  PROC DrawPart12()
    MoveL Offs(pOrigin,259.21,32.84,0.00),v40,z0,tPen\WObj:=wPaper;
    MoveL Offs(pOrigin,259.99,30.50,0.00),v40,z0,tPen\WObj:=wPaper;
    MoveL Offs(pOrigin,259.77,29.44,0.00),v40,z0,tPen\WObj:=wPaper;
    MoveL Offs(pOrigin,259.77,29.44,0.00),v40,z0,tPen\WObj:=wPaper;
    MoveL Offs(pOrigin,257.23,29.30,0.00),v40,z0,tPen\WObj:=wPaper;
    MoveL Offs(pOrigin,255.74,30.50,0.00),v40,z0,tPen\WObj:=wPaper;
    MoveL Offs(pOrigin,255.31,31.35,0.00),v40,z0,tPen\WObj:=wPaper;
    MoveL Offs(pOrigin,255.38,31.99,0.00),v40,z0,tPen\WObj:=wPaper;
    MoveL Offs(pOrigin,256.16,32.84,0.00),v40,z0,tPen\WObj:=wPaper;
    MoveL Offs(pOrigin,257.65,33.83,0.00),v40,z0,tPen\WObj:=wPaper;
    MoveL Offs(pOrigin,258.50,33.90,0.00),v40,z0,tPen\WObj:=wPaper;
    MoveL Offs(pOrigin,257.86,34.01,0.00),v40,z0,tPen\WObj:=wPaper;
    MoveL Offs(pOrigin,256.16,34.01,0.00),v40,z0,tPen\WObj:=wPaper;
    MoveL Offs(pOrigin,256.16,32.95,0.00),v40,z0,tPen\WObj:=wPaper;
    MoveL Offs(pOrigin,254.46,32.95,0.00),v40,z0,tPen\WObj:=wPaper;
    MoveL Offs(pOrigin,254.51,32.62,0.00),v40,z0,tPen\WObj:=wPaper;
    MoveL Offs(pOrigin,254.51,29.86,0.00),v40,z0,tPen\WObj:=wPaper;
    MoveL Offs(pOrigin,254.26,29.05,0.00),v40,z0,tPen\WObj:=wPaper;
    MoveL Offs(pOrigin,255.91,30.70,0.00),v40,z0,tPen\WObj:=wPaper;
    MoveL Offs(pOrigin,255.52,30.84,0.00),v40,z0,tPen\WObj:=wPaper;
    MoveL Offs(pOrigin,245.54,30.84,0.00),v40,z0,tPen\WObj:=wPaper;
    MoveL Offs(pOrigin,245.27,30.52,0.00),v40,z0,tPen\WObj:=wPaper;
    MoveL Offs(pOrigin,246.78,32.02,0.00),v40,z0,tPen\WObj:=wPaper;
    MoveL Offs(pOrigin,246.18,31.90,0.00),v40,z0,tPen\WObj:=wPaper;
    MoveL Offs(pOrigin,244.69,31.90,0.00),v40,z0,tPen\WObj:=wPaper;
    MoveL Offs(pOrigin,244.53,31.26,0.00),v40,z0,tPen\WObj:=wPaper;
    MoveL Offs(pOrigin,246.03,32.77,0.00),v40,z0,tPen\WObj:=wPaper;
    MoveL Offs(pOrigin,245.54,32.95,0.00),v40,z0,tPen\WObj:=wPaper;
    MoveL Offs(pOrigin,244.26,32.95,0.00),v40,z0,tPen\WObj:=wPaper;
    MoveL Offs(pOrigin,243.64,33.36,0.00),v40,z0,tPen\WObj:=wPaper;
    MoveL Offs(pOrigin,259.41,49.14,0.00),v40,z0,tPen\WObj:=wPaper;
    MoveL Offs(pOrigin,259.73,49.65,0.00),v40,z0,tPen\WObj:=wPaper;
    MoveL Offs(pOrigin,261.69,47.70,0.00),v40,z0,tPen\WObj:=wPaper;
    MoveL Offs(pOrigin,261.06,47.79,0.00),v40,z0,tPen\WObj:=wPaper;
    MoveL Offs(pOrigin,266.77,53.50,0.00),v40,z0,tPen\WObj:=wPaper;
    MoveL Offs(pOrigin,266.16,53.68,0.00),v40,z0,tPen\WObj:=wPaper;
    MoveL Offs(pOrigin,268.42,51.42,0.00),v40,z0,tPen\WObj:=wPaper;
    MoveL Offs(pOrigin,268.26,52.01,0.00),v40,z0,tPen\WObj:=wPaper;
    MoveL Offs(pOrigin,274.12,57.87,0.00),v40,z0,tPen\WObj:=wPaper;
    MoveL Offs(pOrigin,273.16,58.30,0.00),v40,z0,tPen\WObj:=wPaper;
    MoveL Offs(pOrigin,272.10,58.30,0.00),v40,z0,tPen\WObj:=wPaper;
    MoveL Offs(pOrigin,272.31,58.76,0.00),v40,z0,tPen\WObj:=wPaper;
    MoveL Offs(pOrigin,272.10,59.19,0.00),v40,z0,tPen\WObj:=wPaper;
    MoveL Offs(pOrigin,272.31,58.76,0.00),v40,z0,tPen\WObj:=wPaper;
    MoveL Offs(pOrigin,272.52,59.35,0.00),v40,z0,tPen\WObj:=wPaper;
    MoveL Offs(pOrigin,271.46,59.35,0.00),v40,z0,tPen\WObj:=wPaper;
    MoveL Offs(pOrigin,271.89,60.41,0.00),v40,z0,tPen\WObj:=wPaper;
    MoveL Offs(pOrigin,270.82,60.41,0.00),v40,z0,tPen\WObj:=wPaper;
    MoveL Offs(pOrigin,271.04,61.10,0.00),v40,z0,tPen\WObj:=wPaper;
    MoveL Offs(pOrigin,272.95,57.49,0.00),v40,z0,tPen\WObj:=wPaper;
    MoveL Offs(pOrigin,272.95,57.49,0.00),v40,z0,tPen\WObj:=wPaper;
    MoveL Offs(pOrigin,272.67,55.58,0.00),v40,z0,tPen\WObj:=wPaper;
    MoveL Offs(pOrigin,271.04,55.43,0.00),v40,z0,tPen\WObj:=wPaper;
    MoveL Offs(pOrigin,268.06,60.46,0.00),v40,z0,tPen\WObj:=wPaper;
    MoveL Offs(pOrigin,268.06,60.46,0.00),v40,z0,tPen\WObj:=wPaper;
    MoveL Offs(pOrigin,268.91,61.53,0.00),v40,z0,tPen\WObj:=wPaper;
    MoveL Offs(pOrigin,270.97,61.31,0.00),v40,z0,tPen\WObj:=wPaper;
    MoveL Offs(pOrigin,271.25,62.59,0.00),v40,z0,tPen\WObj:=wPaper;
    MoveL Offs(pOrigin,276.77,65.28,0.00),v40,z0,tPen\WObj:=wPaper;
    MoveL Offs(pOrigin,281.45,67.05,0.00),v40,z0,tPen\WObj:=wPaper;
    MoveL Offs(pOrigin,283.58,67.26,0.00),v40,z0,tPen\WObj:=wPaper;
    MoveL Offs(pOrigin,286.12,66.48,0.00),v40,z0,tPen\WObj:=wPaper;
    MoveL Offs(pOrigin,292.71,62.94,0.00),v40,z0,tPen\WObj:=wPaper;
    MoveL Offs(pOrigin,300.36,60.46,0.00),v40,z0,tPen\WObj:=wPaper;
    MoveL Offs(pOrigin,304.61,59.61,0.00),v40,z0,tPen\WObj:=wPaper;
    MoveL Offs(pOrigin,312.26,60.25,0.00),v40,z0,tPen\WObj:=wPaper;
    MoveL Offs(pOrigin,315.45,59.47,0.00),v40,z0,tPen\WObj:=wPaper;
    MoveL Offs(pOrigin,317.58,57.49,0.00),v40,z0,tPen\WObj:=wPaper;
    MoveL Offs(pOrigin,320.27,53.45,0.00),v40,z0,tPen\WObj:=wPaper;
    MoveL Offs(pOrigin,320.41,52.60,0.00),v40,z0,tPen\WObj:=wPaper;
    MoveL Offs(pOrigin,321.68,51.54,0.00),v40,z0,tPen\WObj:=wPaper;
    MoveL Offs(pOrigin,322.25,49.20,0.00),v40,z0,tPen\WObj:=wPaper;
    MoveL Offs(pOrigin,322.25,49.20,0.00),v40,z0,tPen\WObj:=wPaper;
    MoveL Offs(pOrigin,322.67,48.35,0.00),v40,z0,tPen\WObj:=wPaper;
    MoveL Offs(pOrigin,322.25,47.92,0.00),v40,z0,tPen\WObj:=wPaper;
    MoveL Offs(pOrigin,322.25,47.92,0.00),v40,z0,tPen\WObj:=wPaper;
    MoveL Offs(pOrigin,322.89,44.53,0.00),v40,z0,tPen\WObj:=wPaper;
    MoveL Offs(pOrigin,322.89,42.40,0.00),v40,z0,tPen\WObj:=wPaper;
    MoveL Offs(pOrigin,322.89,42.40,0.00),v40,z0,tPen\WObj:=wPaper;
    MoveL Offs(pOrigin,323.52,41.76,0.00),v40,z0,tPen\WObj:=wPaper;
    MoveL Offs(pOrigin,323.45,40.70,0.00),v40,z0,tPen\WObj:=wPaper;
    MoveL Offs(pOrigin,322.89,40.28,0.00),v40,z0,tPen\WObj:=wPaper;
    MoveL Offs(pOrigin,322.89,40.28,0.00),v40,z0,tPen\WObj:=wPaper;
    MoveL Offs(pOrigin,322.46,40.70,0.00),v40,z0,tPen\WObj:=wPaper;
    MoveL Offs(pOrigin,322.46,41.97,0.00),v40,z0,tPen\WObj:=wPaper;
    MoveL Offs(pOrigin,322.89,42.40,0.00),v40,z0,tPen\WObj:=wPaper;
    MoveL Offs(pOrigin,322.76,42.29,0.00),v40,z0,tPen\WObj:=wPaper;
    MoveL Offs(pOrigin,324.86,44.39,0.00),v40,z0,tPen\WObj:=wPaper;
    MoveL Offs(pOrigin,325.36,45.25,0.00),v40,z0,tPen\WObj:=wPaper;
    MoveL Offs(pOrigin,319.80,50.81,0.00),v40,fine,tPen\WObj:=wPaper;
    MoveL Offs(pOrigin,319.80,50.81,6.00),v60,z5,tPen\WObj:=wPaper;
    MoveL Offs(pOrigin,321.14,51.12,6.00),vTravel,z5,tPen\WObj:=wPaper;
    MoveL Offs(pOrigin,321.14,51.12,0.00),v60,z0,tPen\WObj:=wPaper;
    MoveL Offs(pOrigin,322.94,52.93,0.00),v40,z0,tPen\WObj:=wPaper;
    MoveL Offs(pOrigin,322.46,53.02,0.00),v40,z0,tPen\WObj:=wPaper;
    MoveL Offs(pOrigin,320.98,53.02,0.00),v40,z0,tPen\WObj:=wPaper;
    MoveL Offs(pOrigin,320.34,52.39,0.00),v40,z0,tPen\WObj:=wPaper;
    MoveL Offs(pOrigin,320.90,50.26,0.00),v40,z0,tPen\WObj:=wPaper;
    MoveL Offs(pOrigin,321.61,49.20,0.00),v40,z0,tPen\WObj:=wPaper;
    MoveL Offs(pOrigin,321.61,49.20,0.00),v40,z0,tPen\WObj:=wPaper;
    MoveL Offs(pOrigin,321.61,48.14,0.00),v40,z0,tPen\WObj:=wPaper;
    MoveL Offs(pOrigin,322.25,47.92,0.00),v40,z0,tPen\WObj:=wPaper;
    MoveL Offs(pOrigin,321.87,47.38,0.00),v40,z0,tPen\WObj:=wPaper;
    MoveL Offs(pOrigin,323.83,49.33,0.00),v40,z0,tPen\WObj:=wPaper;
    MoveL Offs(pOrigin,324.75,48.85,0.00),v40,z0,tPen\WObj:=wPaper;
    MoveL Offs(pOrigin,306.12,67.48,0.00),v40,z0,tPen\WObj:=wPaper;
    MoveL Offs(pOrigin,305.46,66.80,0.00),v40,z0,tPen\WObj:=wPaper;
    MoveL Offs(pOrigin,299.29,60.64,0.00),v40,z0,tPen\WObj:=wPaper;
    MoveL Offs(pOrigin,299.92,61.31,0.00),v40,z0,tPen\WObj:=wPaper;
    MoveL Offs(pOrigin,299.92,63.22,0.00),v40,z0,tPen\WObj:=wPaper;
    MoveL Offs(pOrigin,299.51,63.58,0.00),v40,z0,tPen\WObj:=wPaper;
    MoveL Offs(pOrigin,311.20,63.58,0.00),v40,z0,tPen\WObj:=wPaper;
    MoveL Offs(pOrigin,311.59,63.98,0.00),v40,z0,tPen\WObj:=wPaper;
    MoveL Offs(pOrigin,306.93,59.32,0.00),v40,z0,tPen\WObj:=wPaper;
    MoveL Offs(pOrigin,307.64,58.49,0.00),v40,z0,tPen\WObj:=wPaper;
    MoveL Offs(pOrigin,300.58,65.55,0.00),v40,z0,tPen\WObj:=wPaper;
    MoveL Offs(pOrigin,300.96,65.29,0.00),v40,z0,tPen\WObj:=wPaper;
    MoveL Offs(pOrigin,296.90,61.23,0.00),v40,z0,tPen\WObj:=wPaper;
    MoveL Offs(pOrigin,297.39,61.46,0.00),v40,z0,tPen\WObj:=wPaper;
    MoveL Offs(pOrigin,303.98,61.46,0.00),v40,z0,tPen\WObj:=wPaper;
  ENDPROC

  PROC DrawPart13()
    MoveL Offs(pOrigin,303.34,61.53,0.00),v40,z0,tPen\WObj:=wPaper;
    MoveL Offs(pOrigin,305.89,60.89,0.00),v40,z0,tPen\WObj:=wPaper;
    MoveL Offs(pOrigin,308.86,61.88,0.00),v40,z0,tPen\WObj:=wPaper;
    MoveL Offs(pOrigin,309.29,62.38,0.00),v40,z0,tPen\WObj:=wPaper;
    MoveL Offs(pOrigin,309.29,62.38,0.00),v40,z0,tPen\WObj:=wPaper;
    MoveL Offs(pOrigin,308.65,62.80,0.00),v40,z0,tPen\WObj:=wPaper;
    MoveL Offs(pOrigin,305.67,62.59,0.00),v40,z0,tPen\WObj:=wPaper;
    MoveL Offs(pOrigin,303.76,62.09,0.00),v40,z0,tPen\WObj:=wPaper;
    MoveL Offs(pOrigin,303.34,61.53,0.00),v40,fine,tPen\WObj:=wPaper;
    MoveL Offs(pOrigin,303.34,61.53,6.00),v60,z5,tPen\WObj:=wPaper;
    MoveL Offs(pOrigin,302.03,62.16,6.00),vTravel,z5,tPen\WObj:=wPaper;
    MoveL Offs(pOrigin,302.03,62.16,0.00),v60,z0,tPen\WObj:=wPaper;
    MoveL Offs(pOrigin,302.03,60.89,0.00),v40,z0,tPen\WObj:=wPaper;
    MoveL Offs(pOrigin,301.54,59.90,0.00),v40,z0,tPen\WObj:=wPaper;
    MoveL Offs(pOrigin,309.50,67.86,0.00),v40,z0,tPen\WObj:=wPaper;
    MoveL Offs(pOrigin,309.86,68.22,0.00),v40,z0,tPen\WObj:=wPaper;
    MoveL Offs(pOrigin,312.87,65.22,0.00),v40,z0,tPen\WObj:=wPaper;
    MoveL Offs(pOrigin,312.04,65.92,0.00),v40,z0,tPen\WObj:=wPaper;
    MoveL Offs(pOrigin,317.90,71.78,0.00),v40,z0,tPen\WObj:=wPaper;
    MoveL Offs(pOrigin,317.94,72.09,0.00),v40,z0,tPen\WObj:=wPaper;
    MoveL Offs(pOrigin,325.00,65.03,0.00),v40,z0,tPen\WObj:=wPaper;
    MoveL Offs(pOrigin,325.38,65.82,0.00),v40,z0,tPen\WObj:=wPaper;
    MoveL Offs(pOrigin,326.88,67.32,0.00),v40,z0,tPen\WObj:=wPaper;
    MoveL Offs(pOrigin,326.71,66.74,0.00),v40,z0,tPen\WObj:=wPaper;
    MoveL Offs(pOrigin,323.74,66.74,0.00),v40,z0,tPen\WObj:=wPaper;
    MoveL Offs(pOrigin,324.33,66.26,0.00),v40,z0,tPen\WObj:=wPaper;
    MoveL Offs(pOrigin,325.83,67.76,0.00),v40,z0,tPen\WObj:=wPaper;
    MoveL Offs(pOrigin,326.49,68.02,0.00),v40,z0,tPen\WObj:=wPaper;
    MoveL Offs(pOrigin,349.18,45.33,0.00),v40,z0,tPen\WObj:=wPaper;
    MoveL Offs(pOrigin,348.53,45.66,0.00),v40,z0,tPen\WObj:=wPaper;
    MoveL Offs(pOrigin,347.03,44.16,0.00),v40,z0,tPen\WObj:=wPaper;
    MoveL Offs(pOrigin,347.11,44.53,0.00),v40,z0,tPen\WObj:=wPaper;
    MoveL Offs(pOrigin,346.90,44.95,0.00),v40,z0,tPen\WObj:=wPaper;
    MoveL Offs(pOrigin,347.11,44.53,0.00),v40,z0,tPen\WObj:=wPaper;
    MoveL Offs(pOrigin,347.33,44.57,0.00),v40,z0,tPen\WObj:=wPaper;
    MoveL Offs(pOrigin,348.39,44.57,0.00),v40,z0,tPen\WObj:=wPaper;
    MoveL Offs(pOrigin,348.98,44.62,0.00),v40,z0,tPen\WObj:=wPaper;
    MoveL Offs(pOrigin,347.33,42.96,0.00),v40,z0,tPen\WObj:=wPaper;
    MoveL Offs(pOrigin,347.75,43.51,0.00),v40,z0,tPen\WObj:=wPaper;
    MoveL Offs(pOrigin,349.02,43.51,0.00),v40,z0,tPen\WObj:=wPaper;
    MoveL Offs(pOrigin,349.58,43.72,0.00),v40,z0,tPen\WObj:=wPaper;
    MoveL Offs(pOrigin,347.47,41.62,0.00),v40,z0,tPen\WObj:=wPaper;
    MoveL Offs(pOrigin,347.96,41.40,0.00),v40,z0,tPen\WObj:=wPaper;
    MoveL Offs(pOrigin,349.88,41.40,0.00),v40,z0,tPen\WObj:=wPaper;
    MoveL Offs(pOrigin,349.55,41.34,0.00),v40,z0,tPen\WObj:=wPaper;
    MoveL Offs(pOrigin,349.55,39.00,0.00),v40,z0,tPen\WObj:=wPaper;
    MoveL Offs(pOrigin,349.24,38.36,0.00),v40,z0,tPen\WObj:=wPaper;
    MoveL Offs(pOrigin,349.66,37.72,0.00),v40,z0,tPen\WObj:=wPaper;
    MoveL Offs(pOrigin,349.66,35.60,0.00),v40,z0,tPen\WObj:=wPaper;
    MoveL Offs(pOrigin,348.88,32.41,0.00),v40,z0,tPen\WObj:=wPaper;
    MoveL Offs(pOrigin,346.90,28.80,0.00),v40,z0,tPen\WObj:=wPaper;
    MoveL Offs(pOrigin,345.41,27.31,0.00),v40,z0,tPen\WObj:=wPaper;
    MoveL Offs(pOrigin,343.92,26.39,0.00),v40,z0,tPen\WObj:=wPaper;
    MoveL Offs(pOrigin,341.38,25.61,0.00),v40,z0,tPen\WObj:=wPaper;
    MoveL Offs(pOrigin,339.46,25.83,0.00),v40,z0,tPen\WObj:=wPaper;
    MoveL Offs(pOrigin,336.91,26.67,0.00),v40,z0,tPen\WObj:=wPaper;
    MoveL Offs(pOrigin,336.49,27.10,0.00),v40,z0,tPen\WObj:=wPaper;
    MoveL Offs(pOrigin,336.49,27.10,0.00),v40,z0,tPen\WObj:=wPaper;
    MoveL Offs(pOrigin,337.12,27.52,0.00),v40,z0,tPen\WObj:=wPaper;
    MoveL Offs(pOrigin,340.95,27.10,0.00),v40,z0,tPen\WObj:=wPaper;
    MoveL Offs(pOrigin,343.92,28.38,0.00),v40,z0,tPen\WObj:=wPaper;
    MoveL Offs(pOrigin,346.33,31.35,0.00),v40,z0,tPen\WObj:=wPaper;
    MoveL Offs(pOrigin,347.82,34.54,0.00),v40,z0,tPen\WObj:=wPaper;
    MoveL Offs(pOrigin,348.88,38.15,0.00),v40,z0,tPen\WObj:=wPaper;
    MoveL Offs(pOrigin,349.24,38.36,0.00),v40,z0,tPen\WObj:=wPaper;
    MoveL Offs(pOrigin,348.49,39.00,0.00),v40,z0,tPen\WObj:=wPaper;
    MoveL Offs(pOrigin,348.49,43.25,0.00),v40,z0,tPen\WObj:=wPaper;
    MoveL Offs(pOrigin,347.96,42.46,0.00),v40,z0,tPen\WObj:=wPaper;
    MoveL Offs(pOrigin,349.45,42.46,0.00),v40,z0,tPen\WObj:=wPaper;
    MoveL Offs(pOrigin,350.02,42.67,0.00),v40,z0,tPen\WObj:=wPaper;
    MoveL Offs(pOrigin,347.32,39.97,0.00),v40,z0,tPen\WObj:=wPaper;
    MoveL Offs(pOrigin,346.80,40.25,0.00),v40,z0,tPen\WObj:=wPaper;
    MoveL Offs(pOrigin,351.76,35.29,0.00),v40,z0,tPen\WObj:=wPaper;
    MoveL Offs(pOrigin,351.05,34.74,0.00),v40,z0,tPen\WObj:=wPaper;
    MoveL Offs(pOrigin,348.04,31.73,0.00),v40,z0,tPen\WObj:=wPaper;
    MoveL Offs(pOrigin,347.14,32.33,0.00),v40,z0,tPen\WObj:=wPaper;
    MoveL Offs(pOrigin,339.18,24.36,0.00),v40,z0,tPen\WObj:=wPaper;
    MoveL Offs(pOrigin,339.89,24.50,0.00),v40,z0,tPen\WObj:=wPaper;
    MoveL Offs(pOrigin,346.69,24.50,0.00),v40,z0,tPen\WObj:=wPaper;
    MoveL Offs(pOrigin,346.22,23.94,0.00),v40,z0,tPen\WObj:=wPaper;
    MoveL Offs(pOrigin,349.37,27.09,0.00),v40,z0,tPen\WObj:=wPaper;
    MoveL Offs(pOrigin,350.43,27.65,0.00),v40,z0,tPen\WObj:=wPaper;
    MoveL Offs(pOrigin,352.53,25.55,0.00),v40,z0,tPen\WObj:=wPaper;
    MoveL Offs(pOrigin,353.12,26.35,0.00),v40,z0,tPen\WObj:=wPaper;
    MoveL Offs(pOrigin,357.47,30.71,0.00),v40,z0,tPen\WObj:=wPaper;
    MoveL Offs(pOrigin,357.61,30.92,0.00),v40,z0,tPen\WObj:=wPaper;
    MoveL Offs(pOrigin,359.86,28.67,0.00),v40,z0,tPen\WObj:=wPaper;
    MoveL Offs(pOrigin,358.82,28.22,0.00),v40,z0,tPen\WObj:=wPaper;
    MoveL Offs(pOrigin,356.56,30.48,0.00),v40,z0,tPen\WObj:=wPaper;
    MoveL Offs(pOrigin,355.52,30.03,0.00),v40,z0,tPen\WObj:=wPaper;
    MoveL Offs(pOrigin,357.77,27.78,0.00),v40,z0,tPen\WObj:=wPaper;
    MoveL Offs(pOrigin,357.52,28.73,0.00),v40,z0,tPen\WObj:=wPaper;
    MoveL Offs(pOrigin,355.40,28.73,0.00),v40,z0,tPen\WObj:=wPaper;
    MoveL Offs(pOrigin,354.47,29.20,0.00),v40,z0,tPen\WObj:=wPaper;
    MoveL Offs(pOrigin,350.57,25.30,0.00),v40,z0,tPen\WObj:=wPaper;
    MoveL Offs(pOrigin,350.30,25.56,0.00),v40,z0,tPen\WObj:=wPaper;
    MoveL Offs(pOrigin,341.80,25.56,0.00),v40,fine,tPen\WObj:=wPaper;
    MoveL Offs(pOrigin,341.80,25.56,6.00),v60,z5,tPen\WObj:=wPaper;
    MoveL Offs(pOrigin,342.93,26.62,6.00),vTravel,z5,tPen\WObj:=wPaper;
    MoveL Offs(pOrigin,342.93,26.62,0.00),v60,z0,tPen\WObj:=wPaper;
    MoveL Offs(pOrigin,340.23,23.92,0.00),v40,z0,tPen\WObj:=wPaper;
    MoveL Offs(pOrigin,339.81,23.34,0.00),v40,z0,tPen\WObj:=wPaper;
    MoveL Offs(pOrigin,333.80,29.35,0.00),v40,z0,tPen\WObj:=wPaper;
    MoveL Offs(pOrigin,333.20,28.84,0.00),v40,z0,tPen\WObj:=wPaper;
    MoveL Offs(pOrigin,330.65,26.28,0.00),v40,z0,tPen\WObj:=wPaper;
    MoveL Offs(pOrigin,330.32,26.62,0.00),v40,z0,tPen\WObj:=wPaper;
    MoveL Offs(pOrigin,325.23,26.62,0.00),v40,z0,tPen\WObj:=wPaper;
    MoveL Offs(pOrigin,325.71,27.32,0.00),v40,z0,tPen\WObj:=wPaper;
    MoveL Offs(pOrigin,323.30,24.91,0.00),v40,z0,tPen\WObj:=wPaper;
    MoveL Offs(pOrigin,323.63,24.59,0.00),v40,z0,tPen\WObj:=wPaper;
    MoveL Offs(pOrigin,316.41,31.80,0.00),v40,z0,tPen\WObj:=wPaper;
    MoveL Offs(pOrigin,315.83,30.88,0.00),v40,z0,tPen\WObj:=wPaper;
    MoveL Offs(pOrigin,311.32,26.38,0.00),v40,z0,tPen\WObj:=wPaper;
    MoveL Offs(pOrigin,311.20,26.62,0.00),v40,z0,tPen\WObj:=wPaper;
    MoveL Offs(pOrigin,308.44,26.62,0.00),v40,z0,tPen\WObj:=wPaper;
    MoveL Offs(pOrigin,307.73,27.26,0.00),v40,z0,tPen\WObj:=wPaper;
    MoveL Offs(pOrigin,305.18,24.71,0.00),v40,z0,tPen\WObj:=wPaper;
    MoveL Offs(pOrigin,304.90,23.90,0.00),v40,z0,tPen\WObj:=wPaper;
    MoveL Offs(pOrigin,302.20,26.60,0.00),v40,z0,tPen\WObj:=wPaper;
    MoveL Offs(pOrigin,302.19,26.20,0.00),v40,z0,tPen\WObj:=wPaper;
  ENDPROC

  PROC DrawPart14()
    MoveL Offs(pOrigin,300.23,24.24,0.00),v40,z0,tPen\WObj:=wPaper;
    MoveL Offs(pOrigin,300.71,23.61,0.00),v40,z0,tPen\WObj:=wPaper;
    MoveL Offs(pOrigin,295.75,28.57,0.00),v40,z0,tPen\WObj:=wPaper;
    MoveL Offs(pOrigin,296.35,27.83,0.00),v40,z0,tPen\WObj:=wPaper;
    MoveL Offs(pOrigin,293.34,24.82,0.00),v40,z0,tPen\WObj:=wPaper;
    MoveL Offs(pOrigin,292.77,24.08,0.00),v40,z0,tPen\WObj:=wPaper;
    MoveL Offs(pOrigin,290.21,26.64,0.00),v40,z0,tPen\WObj:=wPaper;
    MoveL Offs(pOrigin,290.20,26.16,0.00),v40,z0,tPen\WObj:=wPaper;
    MoveL Offs(pOrigin,287.35,23.31,0.00),v40,z0,tPen\WObj:=wPaper;
    MoveL Offs(pOrigin,288.13,22.75,0.00),v40,z0,tPen\WObj:=wPaper;
    MoveL Offs(pOrigin,285.42,25.45,0.00),v40,z0,tPen\WObj:=wPaper;
    MoveL Offs(pOrigin,285.85,24.80,0.00),v40,z0,tPen\WObj:=wPaper;
    MoveL Offs(pOrigin,283.75,22.70,0.00),v40,z0,tPen\WObj:=wPaper;
    MoveL Offs(pOrigin,284.24,22.16,0.00),v40,z0,tPen\WObj:=wPaper;
    MoveL Offs(pOrigin,281.38,25.02,0.00),v40,z0,tPen\WObj:=wPaper;
    MoveL Offs(pOrigin,281.06,24.48,0.00),v40,z0,tPen\WObj:=wPaper;
    MoveL Offs(pOrigin,279.26,22.68,0.00),v40,z0,tPen\WObj:=wPaper;
    MoveL Offs(pOrigin,279.89,22.03,0.00),v40,z0,tPen\WObj:=wPaper;
    MoveL Offs(pOrigin,270.73,31.19,0.00),v40,z0,tPen\WObj:=wPaper;
    MoveL Offs(pOrigin,271.04,30.90,0.00),v40,z0,tPen\WObj:=wPaper;
    MoveL Offs(pOrigin,262.03,21.88,0.00),v40,z0,tPen\WObj:=wPaper;
    MoveL Offs(pOrigin,262.47,20.83,0.00),v40,z0,tPen\WObj:=wPaper;
    MoveL Offs(pOrigin,259.47,17.83,0.00),v40,z0,tPen\WObj:=wPaper;
    MoveL Offs(pOrigin,259.77,18.17,0.00),v40,z0,tPen\WObj:=wPaper;
    MoveL Offs(pOrigin,254.68,18.17,0.00),v40,z0,tPen\WObj:=wPaper;
    MoveL Offs(pOrigin,254.38,18.71,0.00),v40,z0,tPen\WObj:=wPaper;
    MoveL Offs(pOrigin,251.37,15.71,0.00),v40,z0,tPen\WObj:=wPaper;
    MoveL Offs(pOrigin,251.15,14.92,0.00),v40,z0,tPen\WObj:=wPaper;
    MoveL Offs(pOrigin,244.24,21.84,0.00),v40,z0,tPen\WObj:=wPaper;
    MoveL Offs(pOrigin,245.25,21.53,0.00),v40,z0,tPen\WObj:=wPaper;
    MoveL Offs(pOrigin,239.39,15.67,0.00),v40,fine,tPen\WObj:=wPaper;
    MoveL Offs(pOrigin,239.39,15.67,6.00),v60,z5,tPen\WObj:=wPaper;
    MoveL Offs(pOrigin,240.58,15.37,6.00),vTravel,z5,tPen\WObj:=wPaper;
    MoveL Offs(pOrigin,240.58,15.37,0.00),v60,z0,tPen\WObj:=wPaper;
    MoveL Offs(pOrigin,237.13,11.92,0.00),v40,z0,tPen\WObj:=wPaper;
    MoveL Offs(pOrigin,236.82,11.83,0.00),v40,z0,tPen\WObj:=wPaper;
    MoveL Offs(pOrigin,226.84,11.83,0.00),v40,z0,tPen\WObj:=wPaper;
    MoveL Offs(pOrigin,226.64,11.88,0.00),v40,z0,tPen\WObj:=wPaper;
    MoveL Offs(pOrigin,230.70,15.94,0.00),v40,z0,tPen\WObj:=wPaper;
    MoveL Offs(pOrigin,230.88,15.00,0.00),v40,z0,tPen\WObj:=wPaper;
    MoveL Offs(pOrigin,228.32,15.00,0.00),v40,z0,tPen\WObj:=wPaper;
    MoveL Offs(pOrigin,227.85,16.08,0.00),v40,z0,tPen\WObj:=wPaper;
    MoveL Offs(pOrigin,223.80,12.03,0.00),v40,z0,tPen\WObj:=wPaper;
    MoveL Offs(pOrigin,223.30,11.41,0.00),v40,z0,tPen\WObj:=wPaper;
    MoveL Offs(pOrigin,212.33,22.38,0.00),v40,z0,tPen\WObj:=wPaper;
    MoveL Offs(pOrigin,213.04,22.18,0.00),v40,z0,tPen\WObj:=wPaper;
    MoveL Offs(pOrigin,204.33,13.46,0.00),v40,z0,tPen\WObj:=wPaper;
    MoveL Offs(pOrigin,204.27,12.52,0.00),v40,z0,tPen\WObj:=wPaper;
    MoveL Offs(pOrigin,200.07,16.73,0.00),v40,z0,tPen\WObj:=wPaper;
    MoveL Offs(pOrigin,199.54,16.15,0.00),v40,z0,tPen\WObj:=wPaper;
    MoveL Offs(pOrigin,197.44,14.04,0.00),v40,z0,tPen\WObj:=wPaper;
    MoveL Offs(pOrigin,197.94,13.94,0.00),v40,z0,tPen\WObj:=wPaper;
    MoveL Offs(pOrigin,221.31,13.94,0.00),v40,fine,tPen\WObj:=wPaper;
    MoveL Offs(pOrigin,221.31,13.94,6.00),v60,z5,tPen\WObj:=wPaper;
    MoveL Offs(pOrigin,222.60,12.32,6.00),vTravel,z5,tPen\WObj:=wPaper;
    MoveL Offs(pOrigin,222.60,12.32,0.00),v60,z0,tPen\WObj:=wPaper;
    MoveL Offs(pOrigin,226.66,16.38,0.00),v40,fine,tPen\WObj:=wPaper;
    MoveL Offs(pOrigin,226.66,16.38,6.00),v60,z5,tPen\WObj:=wPaper;
    MoveL Offs(pOrigin,226.51,17.73,6.00),vTravel,z5,tPen\WObj:=wPaper;
    MoveL Offs(pOrigin,226.51,17.73,0.00),v60,z0,tPen\WObj:=wPaper;
    MoveL Offs(pOrigin,227.86,19.08,0.00),v40,z0,tPen\WObj:=wPaper;
    MoveL Offs(pOrigin,228.67,19.49,0.00),v40,z0,tPen\WObj:=wPaper;
    MoveL Offs(pOrigin,236.93,11.22,0.00),v40,fine,tPen\WObj:=wPaper;
    MoveL Offs(pOrigin,236.93,11.22,6.00),v60,z5,tPen\WObj:=wPaper;
    MoveL Offs(pOrigin,238.28,11.37,6.00),vTravel,z5,tPen\WObj:=wPaper;
    MoveL Offs(pOrigin,238.28,11.37,0.00),v60,z0,tPen\WObj:=wPaper;
    MoveL Offs(pOrigin,230.32,19.33,0.00),v40,z0,tPen\WObj:=wPaper;
    MoveL Offs(pOrigin,230.71,18.94,0.00),v40,z0,tPen\WObj:=wPaper;
    MoveL Offs(pOrigin,229.06,17.28,0.00),v40,fine,tPen\WObj:=wPaper;
    MoveL Offs(pOrigin,229.06,17.28,6.00),v60,z5,tPen\WObj:=wPaper;
    MoveL Offs(pOrigin,227.86,17.58,6.00),vTravel,z5,tPen\WObj:=wPaper;
    MoveL Offs(pOrigin,227.86,17.58,0.00),v60,z0,tPen\WObj:=wPaper;
    MoveL Offs(pOrigin,229.36,19.08,0.00),v40,fine,tPen\WObj:=wPaper;
    MoveL Offs(pOrigin,229.36,19.08,6.00),v60,z5,tPen\WObj:=wPaper;
    MoveL Offs(pOrigin,230.40,17.14,6.00),vTravel,z5,tPen\WObj:=wPaper;
    MoveL Offs(pOrigin,230.40,17.14,0.00),v60,z0,tPen\WObj:=wPaper;
    MoveL Offs(pOrigin,232.21,18.94,0.00),v40,z0,tPen\WObj:=wPaper;
    MoveL Offs(pOrigin,231.81,19.33,0.00),v40,z0,tPen\WObj:=wPaper;
    MoveL Offs(pOrigin,239.33,11.81,0.00),v40,z0,tPen\WObj:=wPaper;
    MoveL Offs(pOrigin,239.23,12.52,0.00),v40,z0,tPen\WObj:=wPaper;
    MoveL Offs(pOrigin,242.53,15.83,0.00),v40,z0,tPen\WObj:=wPaper;
    MoveL Offs(pOrigin,242.99,15.00,0.00),v40,z0,tPen\WObj:=wPaper;
    MoveL Offs(pOrigin,248.72,15.00,0.00),v40,z0,tPen\WObj:=wPaper;
    MoveL Offs(pOrigin,249.27,15.10,0.00),v40,z0,tPen\WObj:=wPaper;
    MoveL Offs(pOrigin,252.58,18.41,0.00),v40,z0,tPen\WObj:=wPaper;
    MoveL Offs(pOrigin,251.98,19.30,0.00),v40,z0,tPen\WObj:=wPaper;
    MoveL Offs(pOrigin,257.24,24.56,0.00),v40,z0,tPen\WObj:=wPaper;
    MoveL Offs(pOrigin,257.56,24.94,0.00),v40,z0,tPen\WObj:=wPaper;
    MoveL Offs(pOrigin,264.17,18.33,0.00),v40,z0,tPen\WObj:=wPaper;
    MoveL Offs(pOrigin,263.36,18.74,0.00),v40,z0,tPen\WObj:=wPaper;
    MoveL Offs(pOrigin,266.52,21.89,0.00),v40,z0,tPen\WObj:=wPaper;
    MoveL Offs(pOrigin,266.58,21.34,0.00),v40,z0,tPen\WObj:=wPaper;
    MoveL Offs(pOrigin,271.68,21.34,0.00),v40,z0,tPen\WObj:=wPaper;
    MoveL Offs(pOrigin,271.46,20.86,0.00),v40,z0,tPen\WObj:=wPaper;
    MoveL Offs(pOrigin,276.42,25.82,0.00),v40,z0,tPen\WObj:=wPaper;
    MoveL Offs(pOrigin,276.58,26.83,0.00),v40,z0,tPen\WObj:=wPaper;
    MoveL Offs(pOrigin,272.07,31.34,0.00),v40,z0,tPen\WObj:=wPaper;
    MoveL Offs(pOrigin,272.46,30.29,0.00),v40,z0,tPen\WObj:=wPaper;
    MoveL Offs(pOrigin,272.46,27.95,0.00),v40,fine,tPen\WObj:=wPaper;
    MoveL Offs(pOrigin,272.46,27.95,6.00),v60,z5,tPen\WObj:=wPaper;
    MoveL Offs(pOrigin,273.52,27.10,6.00),vTravel,z5,tPen\WObj:=wPaper;
    MoveL Offs(pOrigin,273.52,27.10,0.00),v60,z0,tPen\WObj:=wPaper;
    MoveL Offs(pOrigin,273.52,30.50,0.00),v40,z0,tPen\WObj:=wPaper;
    MoveL Offs(pOrigin,273.38,30.84,0.00),v40,z0,tPen\WObj:=wPaper;
    MoveL Offs(pOrigin,276.77,30.84,0.00),v40,z0,tPen\WObj:=wPaper;
    MoveL Offs(pOrigin,276.43,30.31,0.00),v40,z0,tPen\WObj:=wPaper;
    MoveL Offs(pOrigin,279.44,33.32,0.00),v40,z0,tPen\WObj:=wPaper;
    MoveL Offs(pOrigin,279.86,34.01,0.00),v40,z0,tPen\WObj:=wPaper;
    MoveL Offs(pOrigin,282.11,31.76,0.00),v40,z0,tPen\WObj:=wPaper;
    MoveL Offs(pOrigin,281.08,31.97,0.00),v40,z0,tPen\WObj:=wPaper;
    MoveL Offs(pOrigin,288.74,39.64,0.00),v40,z0,tPen\WObj:=wPaper;
    MoveL Offs(pOrigin,288.00,40.38,0.00),v40,z0,tPen\WObj:=wPaper;
    MoveL Offs(pOrigin,285.44,37.83,0.00),v40,z0,tPen\WObj:=wPaper;
    MoveL Offs(pOrigin,284.49,38.34,0.00),v40,z0,tPen\WObj:=wPaper;
    MoveL Offs(pOrigin,288.39,34.43,0.00),v40,z0,tPen\WObj:=wPaper;
    MoveL Offs(pOrigin,288.73,35.14,0.00),v40,z0,tPen\WObj:=wPaper;
    MoveL Offs(pOrigin,292.49,38.90,0.00),v40,z0,tPen\WObj:=wPaper;
    MoveL Offs(pOrigin,291.86,38.36,0.00),v40,z0,tPen\WObj:=wPaper;
    MoveL Offs(pOrigin,291.08,38.58,0.00),v40,z0,tPen\WObj:=wPaper;
    MoveL Offs(pOrigin,291.01,39.21,0.00),v40,z0,tPen\WObj:=wPaper;
  ENDPROC

  PROC DrawPart15()
    MoveL Offs(pOrigin,291.23,39.57,0.00),v40,z0,tPen\WObj:=wPaper;
    MoveL Offs(pOrigin,291.86,39.64,0.00),v40,z0,tPen\WObj:=wPaper;
    MoveL Offs(pOrigin,291.86,39.64,0.00),v40,z0,tPen\WObj:=wPaper;
    MoveL Offs(pOrigin,291.37,42.19,0.00),v40,z0,tPen\WObj:=wPaper;
    MoveL Offs(pOrigin,290.38,42.83,0.00),v40,z0,tPen\WObj:=wPaper;
    MoveL Offs(pOrigin,290.09,42.61,0.00),v40,z0,tPen\WObj:=wPaper;
    MoveL Offs(pOrigin,290.16,40.49,0.00),v40,z0,tPen\WObj:=wPaper;
    MoveL Offs(pOrigin,290.16,40.49,0.00),v40,z0,tPen\WObj:=wPaper;
    MoveL Offs(pOrigin,287.19,40.49,0.00),v40,z0,tPen\WObj:=wPaper;
    MoveL Offs(pOrigin,287.19,40.49,0.00),v40,z0,tPen\WObj:=wPaper;
    MoveL Offs(pOrigin,287.19,39.42,0.00),v40,z0,tPen\WObj:=wPaper;
    MoveL Offs(pOrigin,287.19,39.42,0.00),v40,z0,tPen\WObj:=wPaper;
    MoveL Offs(pOrigin,288.25,38.79,0.00),v40,z0,tPen\WObj:=wPaper;
    MoveL Offs(pOrigin,289.74,39.21,0.00),v40,z0,tPen\WObj:=wPaper;
    MoveL Offs(pOrigin,289.74,39.21,0.00),v40,z0,tPen\WObj:=wPaper;
    MoveL Offs(pOrigin,290.38,39.85,0.00),v40,z0,tPen\WObj:=wPaper;
    MoveL Offs(pOrigin,289.65,40.54,0.00),v40,z0,tPen\WObj:=wPaper;
    MoveL Offs(pOrigin,291.45,42.34,0.00),v40,z0,tPen\WObj:=wPaper;
    MoveL Offs(pOrigin,291.81,42.96,0.00),v40,z0,tPen\WObj:=wPaper;
    MoveL Offs(pOrigin,285.80,48.97,0.00),v40,z0,tPen\WObj:=wPaper;
    MoveL Offs(pOrigin,285.63,48.47,0.00),v40,z0,tPen\WObj:=wPaper;
    MoveL Offs(pOrigin,282.02,44.86,0.00),v40,fine,tPen\WObj:=wPaper;
    MoveL Offs(pOrigin,282.02,44.86,6.00),v60,z5,tPen\WObj:=wPaper;
    MoveL Offs(pOrigin,280.52,44.86,6.00),vTravel,z5,tPen\WObj:=wPaper;
    MoveL Offs(pOrigin,280.52,44.86,0.00),v60,z0,tPen\WObj:=wPaper;
    MoveL Offs(pOrigin,283.38,47.71,0.00),v40,z0,tPen\WObj:=wPaper;
    MoveL Offs(pOrigin,283.71,48.08,0.00),v40,z0,tPen\WObj:=wPaper;
    MoveL Offs(pOrigin,294.83,36.96,0.00),v40,z0,tPen\WObj:=wPaper;
    MoveL Offs(pOrigin,295.42,37.86,0.00),v40,z0,tPen\WObj:=wPaper;
    MoveL Offs(pOrigin,294.07,39.21,0.00),v40,z0,tPen\WObj:=wPaper;
    MoveL Offs(pOrigin,293.53,38.45,0.00),v40,z0,tPen\WObj:=wPaper;
    MoveL Offs(pOrigin,291.28,36.20,0.00),v40,z0,tPen\WObj:=wPaper;
    MoveL Offs(pOrigin,291.68,35.62,0.00),v40,z0,tPen\WObj:=wPaper;
    MoveL Offs(pOrigin,280.26,47.04,0.00),v40,z0,tPen\WObj:=wPaper;
    MoveL Offs(pOrigin,281.13,46.95,0.00),v40,z0,tPen\WObj:=wPaper;
    MoveL Offs(pOrigin,278.12,43.95,0.00),v40,z0,tPen\WObj:=wPaper;
    MoveL Offs(pOrigin,278.18,43.15,0.00),v40,z0,tPen\WObj:=wPaper;
    MoveL Offs(pOrigin,275.78,45.56,0.00),v40,z0,tPen\WObj:=wPaper;
    MoveL Offs(pOrigin,276.78,45.59,0.00),v40,z0,tPen\WObj:=wPaper;
    MoveL Offs(pOrigin,272.57,41.39,0.00),v40,z0,tPen\WObj:=wPaper;
    MoveL Offs(pOrigin,272.10,41.40,0.00),v40,z0,tPen\WObj:=wPaper;
    MoveL Offs(pOrigin,270.19,41.40,0.00),v40,z0,tPen\WObj:=wPaper;
    MoveL Offs(pOrigin,269.98,40.34,0.00),v40,z0,tPen\WObj:=wPaper;
    MoveL Offs(pOrigin,268.06,40.34,0.00),v40,z0,tPen\WObj:=wPaper;
    MoveL Offs(pOrigin,267.93,41.22,0.00),v40,z0,tPen\WObj:=wPaper;
    MoveL Offs(pOrigin,263.87,37.17,0.00),v40,z0,tPen\WObj:=wPaper;
    MoveL Offs(pOrigin,263.39,37.18,0.00),v40,z0,tPen\WObj:=wPaper;
    MoveL Offs(pOrigin,261.48,37.18,0.00),v40,z0,tPen\WObj:=wPaper;
    MoveL Offs(pOrigin,261.26,36.12,0.00),v40,z0,tPen\WObj:=wPaper;
    MoveL Offs(pOrigin,259.35,36.12,0.00),v40,z0,tPen\WObj:=wPaper;
    MoveL Offs(pOrigin,259.08,36.85,0.00),v40,z0,tPen\WObj:=wPaper;
    MoveL Offs(pOrigin,250.81,28.59,0.00),v40,z0,tPen\WObj:=wPaper;
    MoveL Offs(pOrigin,251.41,28.10,0.00),v40,z0,tPen\WObj:=wPaper;
    MoveL Offs(pOrigin,237.59,41.93,0.00),v40,z0,tPen\WObj:=wPaper;
    MoveL Offs(pOrigin,238.57,41.73,0.00),v40,z0,tPen\WObj:=wPaper;
    MoveL Offs(pOrigin,235.86,39.03,0.00),v40,z0,tPen\WObj:=wPaper;
    MoveL Offs(pOrigin,235.12,39.29,0.00),v40,z0,tPen\WObj:=wPaper;
    MoveL Offs(pOrigin,243.20,39.29,0.00),v40,z0,tPen\WObj:=wPaper;
    MoveL Offs(pOrigin,242.89,39.64,0.00),v40,z0,tPen\WObj:=wPaper;
    MoveL Offs(pOrigin,242.89,40.70,0.00),v40,z0,tPen\WObj:=wPaper;
    MoveL Offs(pOrigin,242.99,41.40,0.00),v40,z0,tPen\WObj:=wPaper;
    MoveL Offs(pOrigin,244.90,41.40,0.00),v40,z0,tPen\WObj:=wPaper;
    MoveL Offs(pOrigin,244.26,40.91,0.00),v40,z0,tPen\WObj:=wPaper;
    MoveL Offs(pOrigin,245.54,41.97,0.00),v40,z0,tPen\WObj:=wPaper;
    MoveL Offs(pOrigin,245.54,41.97,0.00),v40,z0,tPen\WObj:=wPaper;
    MoveL Offs(pOrigin,243.62,39.85,0.00),v40,z0,tPen\WObj:=wPaper;
    MoveL Offs(pOrigin,242.77,38.15,0.00),v40,z0,tPen\WObj:=wPaper;
    MoveL Offs(pOrigin,242.92,36.66,0.00),v40,z0,tPen\WObj:=wPaper;
    MoveL Offs(pOrigin,243.62,35.67,0.00),v40,z0,tPen\WObj:=wPaper;
    MoveL Offs(pOrigin,244.26,35.81,0.00),v40,z0,tPen\WObj:=wPaper;
    MoveL Offs(pOrigin,245.54,37.72,0.00),v40,z0,tPen\WObj:=wPaper;
    MoveL Offs(pOrigin,247.45,39.42,0.00),v40,z0,tPen\WObj:=wPaper;
    MoveL Offs(pOrigin,247.88,40.28,0.00),v40,z0,tPen\WObj:=wPaper;
    MoveL Offs(pOrigin,248.94,40.34,0.00),v40,z0,tPen\WObj:=wPaper;
    MoveL Offs(pOrigin,250.42,40.34,0.00),v40,z0,tPen\WObj:=wPaper;
    MoveL Offs(pOrigin,250.00,39.85,0.00),v40,z0,tPen\WObj:=wPaper;
    MoveL Offs(pOrigin,250.43,40.28,0.00),v40,z0,tPen\WObj:=wPaper;
    MoveL Offs(pOrigin,250.00,39.85,0.00),v40,z0,tPen\WObj:=wPaper;
    MoveL Offs(pOrigin,250.63,39.34,0.00),v40,z0,tPen\WObj:=wPaper;
    MoveL Offs(pOrigin,248.52,41.45,0.00),v40,z0,tPen\WObj:=wPaper;
    MoveL Offs(pOrigin,248.94,40.49,0.00),v40,z0,tPen\WObj:=wPaper;
    MoveL Offs(pOrigin,249.36,40.91,0.00),v40,z0,tPen\WObj:=wPaper;
    MoveL Offs(pOrigin,248.94,40.49,0.00),v40,fine,tPen\WObj:=wPaper;
    MoveL Offs(pOrigin,248.94,40.49,6.00),v60,z5,tPen\WObj:=wPaper;
    MoveL Offs(pOrigin,250.21,41.40,6.00),vTravel,z5,tPen\WObj:=wPaper;
    MoveL Offs(pOrigin,250.21,41.40,0.00),v60,z0,tPen\WObj:=wPaper;
    MoveL Offs(pOrigin,251.91,41.40,0.00),v40,z0,tPen\WObj:=wPaper;
    MoveL Offs(pOrigin,252.55,41.76,0.00),v40,z0,tPen\WObj:=wPaper;
    MoveL Offs(pOrigin,252.98,42.19,0.00),v40,z0,tPen\WObj:=wPaper;
    MoveL Offs(pOrigin,252.55,41.76,0.00),v40,z0,tPen\WObj:=wPaper;
    MoveL Offs(pOrigin,253.19,42.46,0.00),v40,z0,tPen\WObj:=wPaper;
    MoveL Offs(pOrigin,251.49,42.46,0.00),v40,z0,tPen\WObj:=wPaper;
    MoveL Offs(pOrigin,251.27,42.40,0.00),v40,z0,tPen\WObj:=wPaper;
    MoveL Offs(pOrigin,251.70,42.83,0.00),v40,z0,tPen\WObj:=wPaper;
    MoveL Offs(pOrigin,251.27,42.40,0.00),v40,z0,tPen\WObj:=wPaper;
    MoveL Offs(pOrigin,251.07,43.39,0.00),v40,z0,tPen\WObj:=wPaper;
    MoveL Offs(pOrigin,253.32,41.13,0.00),v40,z0,tPen\WObj:=wPaper;
    MoveL Offs(pOrigin,253.92,42.03,0.00),v40,z0,tPen\WObj:=wPaper;
    MoveL Offs(pOrigin,251.81,44.13,0.00),v40,z0,tPen\WObj:=wPaper;
    MoveL Offs(pOrigin,252.86,44.58,0.00),v40,z0,tPen\WObj:=wPaper;
    MoveL Offs(pOrigin,254.81,42.63,0.00),v40,z0,tPen\WObj:=wPaper;
    MoveL Offs(pOrigin,254.46,43.25,0.00),v40,z0,tPen\WObj:=wPaper;
    MoveL Offs(pOrigin,254.89,43.67,0.00),v40,z0,tPen\WObj:=wPaper;
    MoveL Offs(pOrigin,254.46,43.25,0.00),v40,z0,tPen\WObj:=wPaper;
    MoveL Offs(pOrigin,254.46,43.51,0.00),v40,z0,tPen\WObj:=wPaper;
    MoveL Offs(pOrigin,252.98,43.51,0.00),v40,fine,tPen\WObj:=wPaper;
    MoveL Offs(pOrigin,252.98,43.51,6.00),v60,z5,tPen\WObj:=wPaper;
    MoveL Offs(pOrigin,254.46,44.57,6.00),vTravel,z5,tPen\WObj:=wPaper;
    MoveL Offs(pOrigin,254.46,44.57,0.00),v60,z0,tPen\WObj:=wPaper;
    MoveL Offs(pOrigin,255.95,44.57,0.00),v40,z0,tPen\WObj:=wPaper;
    MoveL Offs(pOrigin,255.65,43.88,0.00),v40,z0,tPen\WObj:=wPaper;
    MoveL Offs(pOrigin,263.62,51.84,0.00),v40,z0,tPen\WObj:=wPaper;
    MoveL Offs(pOrigin,263.17,52.19,0.00),v40,z0,tPen\WObj:=wPaper;
    MoveL Offs(pOrigin,265.43,49.93,0.00),v40,z0,tPen\WObj:=wPaper;
    MoveL Offs(pOrigin,265.11,50.35,0.00),v40,z0,tPen\WObj:=wPaper;
    MoveL Offs(pOrigin,273.67,58.92,0.00),v40,z0,tPen\WObj:=wPaper;
    MoveL Offs(pOrigin,273.94,59.34,0.00),v40,z0,tPen\WObj:=wPaper;
    MoveL Offs(pOrigin,269.13,64.15,0.00),v40,z0,tPen\WObj:=wPaper;
    MoveL Offs(pOrigin,269.95,64.15,0.00),v40,z0,tPen\WObj:=wPaper;
    MoveL Offs(pOrigin,265.59,59.79,0.00),v40,z0,tPen\WObj:=wPaper;
  ENDPROC

  PROC DrawPart16()
    MoveL Offs(pOrigin,265.25,59.07,0.00),v40,z0,tPen\WObj:=wPaper;
    MoveL Offs(pOrigin,262.84,61.48,0.00),v40,z0,tPen\WObj:=wPaper;
    MoveL Offs(pOrigin,262.96,60.41,0.00),v40,z0,tPen\WObj:=wPaper;
    MoveL Offs(pOrigin,268.27,60.41,0.00),v40,z0,tPen\WObj:=wPaper;
    MoveL Offs(pOrigin,268.06,60.46,0.00),v40,z0,tPen\WObj:=wPaper;
    MoveL Offs(pOrigin,265.09,60.11,0.00),v40,z0,tPen\WObj:=wPaper;
    MoveL Offs(pOrigin,259.35,56.85,0.00),v40,z0,tPen\WObj:=wPaper;
    MoveL Offs(pOrigin,250.85,48.78,0.00),v40,z0,tPen\WObj:=wPaper;
    MoveL Offs(pOrigin,246.18,43.46,0.00),v40,z0,tPen\WObj:=wPaper;
    MoveL Offs(pOrigin,245.61,42.19,0.00),v40,z0,tPen\WObj:=wPaper;
    MoveL Offs(pOrigin,247.24,41.34,0.00),v40,z0,tPen\WObj:=wPaper;
    MoveL Offs(pOrigin,248.09,40.35,0.00),v40,z0,tPen\WObj:=wPaper;
    MoveL Offs(pOrigin,248.51,40.42,0.00),v40,z0,tPen\WObj:=wPaper;
    MoveL Offs(pOrigin,260.20,49.20,0.00),v40,z0,tPen\WObj:=wPaper;
    MoveL Offs(pOrigin,264.66,52.03,0.00),v40,z0,tPen\WObj:=wPaper;
    MoveL Offs(pOrigin,269.55,54.16,0.00),v40,z0,tPen\WObj:=wPaper;
    MoveL Offs(pOrigin,270.61,55.58,0.00),v40,z0,tPen\WObj:=wPaper;
    MoveL Offs(pOrigin,271.04,56.18,0.00),v40,z0,tPen\WObj:=wPaper;
    MoveL Offs(pOrigin,269.98,56.18,0.00),v40,z0,tPen\WObj:=wPaper;
    MoveL Offs(pOrigin,269.17,55.91,0.00),v40,z0,tPen\WObj:=wPaper;
    MoveL Offs(pOrigin,273.08,59.81,0.00),v40,z0,tPen\WObj:=wPaper;
    MoveL Offs(pOrigin,272.48,60.71,0.00),v40,z0,tPen\WObj:=wPaper;
    MoveL Offs(pOrigin,268.87,57.10,0.00),v40,z0,tPen\WObj:=wPaper;
    MoveL Offs(pOrigin,269.34,57.24,0.00),v40,z0,tPen\WObj:=wPaper;
    MoveL Offs(pOrigin,270.40,57.24,0.00),v40,z0,tPen\WObj:=wPaper;
    MoveL Offs(pOrigin,269.76,57.49,0.00),v40,z0,tPen\WObj:=wPaper;
    MoveL Offs(pOrigin,269.55,57.91,0.00),v40,z0,tPen\WObj:=wPaper;
    MoveL Offs(pOrigin,269.76,57.49,0.00),v40,z0,tPen\WObj:=wPaper;
    MoveL Offs(pOrigin,269.76,58.30,0.00),v40,z0,tPen\WObj:=wPaper;
    MoveL Offs(pOrigin,268.70,58.30,0.00),v40,z0,tPen\WObj:=wPaper;
    MoveL Offs(pOrigin,268.28,58.00,0.00),v40,z0,tPen\WObj:=wPaper;
    MoveL Offs(pOrigin,272.03,61.76,0.00),v40,z0,tPen\WObj:=wPaper;
    MoveL Offs(pOrigin,271.46,61.46,0.00),v40,z0,tPen\WObj:=wPaper;
    MoveL Offs(pOrigin,265.30,61.46,0.00),v40,fine,tPen\WObj:=wPaper;
    MoveL Offs(pOrigin,265.30,61.46,6.00),v60,z5,tPen\WObj:=wPaper;
    MoveL Offs(pOrigin,263.89,61.92,6.00),vTravel,z5,tPen\WObj:=wPaper;
    MoveL Offs(pOrigin,263.89,61.92,0.00),v60,z0,tPen\WObj:=wPaper;
    MoveL Offs(pOrigin,272.76,53.06,0.00),v40,z0,tPen\WObj:=wPaper;
    MoveL Offs(pOrigin,272.31,54.07,0.00),v40,z0,tPen\WObj:=wPaper;
    MoveL Offs(pOrigin,269.55,54.07,0.00),v40,z0,tPen\WObj:=wPaper;
    MoveL Offs(pOrigin,269.34,53.02,0.00),v40,z0,tPen\WObj:=wPaper;
    MoveL Offs(pOrigin,267.21,53.02,0.00),v40,z0,tPen\WObj:=wPaper;
    MoveL Offs(pOrigin,267.00,51.96,0.00),v40,z0,tPen\WObj:=wPaper;
    MoveL Offs(pOrigin,265.09,51.96,0.00),v40,z0,tPen\WObj:=wPaper;
    MoveL Offs(pOrigin,265.30,50.90,0.00),v40,z0,tPen\WObj:=wPaper;
    MoveL Offs(pOrigin,263.60,50.90,0.00),v40,z0,tPen\WObj:=wPaper;
    MoveL Offs(pOrigin,263.60,49.85,0.00),v40,z0,tPen\WObj:=wPaper;
    MoveL Offs(pOrigin,261.90,49.85,0.00),v40,z0,tPen\WObj:=wPaper;
    MoveL Offs(pOrigin,261.90,48.79,0.00),v40,z0,tPen\WObj:=wPaper;
    MoveL Offs(pOrigin,260.41,48.79,0.00),v40,z0,tPen\WObj:=wPaper;
    MoveL Offs(pOrigin,260.41,47.74,0.00),v40,z0,tPen\WObj:=wPaper;
    MoveL Offs(pOrigin,258.71,47.74,0.00),v40,z0,tPen\WObj:=wPaper;
    MoveL Offs(pOrigin,257.86,47.29,0.00),v40,z0,tPen\WObj:=wPaper;
    MoveL Offs(pOrigin,258.29,47.71,0.00),v40,z0,tPen\WObj:=wPaper;
    MoveL Offs(pOrigin,257.86,47.29,0.00),v40,z0,tPen\WObj:=wPaper;
    MoveL Offs(pOrigin,257.23,46.68,0.00),v40,z0,tPen\WObj:=wPaper;
    MoveL Offs(pOrigin,258.92,46.68,0.00),v40,z0,tPen\WObj:=wPaper;
    MoveL Offs(pOrigin,259.15,45.76,0.00),v40,z0,tPen\WObj:=wPaper;
    MoveL Offs(pOrigin,256.89,48.01,0.00),v40,z0,tPen\WObj:=wPaper;
    MoveL Offs(pOrigin,256.15,47.26,0.00),v40,z0,tPen\WObj:=wPaper;
    MoveL Offs(pOrigin,258.25,45.16,0.00),v40,z0,tPen\WObj:=wPaper;
    MoveL Offs(pOrigin,257.44,45.62,0.00),v40,z0,tPen\WObj:=wPaper;
    MoveL Offs(pOrigin,255.95,45.62,0.00),v40,fine,tPen\WObj:=wPaper;
    MoveL Offs(pOrigin,255.95,45.62,6.00),v60,z5,tPen\WObj:=wPaper;
    MoveL Offs(pOrigin,255.25,46.67,6.00),vTravel,z5,tPen\WObj:=wPaper;
    MoveL Offs(pOrigin,255.25,46.67,0.00),v60,z0,tPen\WObj:=wPaper;
    MoveL Offs(pOrigin,257.50,44.41,0.00),v40,z0,tPen\WObj:=wPaper;
    MoveL Offs(pOrigin,256.61,43.82,0.00),v40,z0,tPen\WObj:=wPaper;
    MoveL Offs(pOrigin,254.35,46.07,0.00),v40,z0,tPen\WObj:=wPaper;
    MoveL Offs(pOrigin,254.31,45.52,0.00),v40,z0,tPen\WObj:=wPaper;
    MoveL Offs(pOrigin,242.89,34.10,0.00),v40,z0,tPen\WObj:=wPaper;
    MoveL Offs(pOrigin,243.41,34.01,0.00),v40,z0,tPen\WObj:=wPaper;
    MoveL Offs(pOrigin,245.32,34.01,0.00),v40,z0,tPen\WObj:=wPaper;
    MoveL Offs(pOrigin,245.73,33.96,0.00),v40,z0,tPen\WObj:=wPaper;
    MoveL Offs(pOrigin,243.93,32.16,0.00),v40,z0,tPen\WObj:=wPaper;
    MoveL Offs(pOrigin,243.91,31.12,0.00),v40,z0,tPen\WObj:=wPaper;
    MoveL Offs(pOrigin,247.67,27.37,0.00),v40,z0,tPen\WObj:=wPaper;
    MoveL Offs(pOrigin,247.51,28.28,0.00),v40,z0,tPen\WObj:=wPaper;
    MoveL Offs(pOrigin,251.27,32.03,0.00),v40,z0,tPen\WObj:=wPaper;
    MoveL Offs(pOrigin,251.34,31.14,0.00),v40,z0,tPen\WObj:=wPaper;
    MoveL Offs(pOrigin,251.34,29.65,0.00),v40,z0,tPen\WObj:=wPaper;
    MoveL Offs(pOrigin,251.91,29.23,0.00),v40,z0,tPen\WObj:=wPaper;
    MoveL Offs(pOrigin,251.06,29.01,0.00),v40,z0,tPen\WObj:=wPaper;
    MoveL Offs(pOrigin,250.64,29.44,0.00),v40,z0,tPen\WObj:=wPaper;
    MoveL Offs(pOrigin,250.64,29.44,0.00),v40,z0,tPen\WObj:=wPaper;
    MoveL Offs(pOrigin,251.06,30.08,0.00),v40,z0,tPen\WObj:=wPaper;
    MoveL Offs(pOrigin,251.91,30.08,0.00),v40,fine,tPen\WObj:=wPaper;
    MoveL Offs(pOrigin,251.91,30.08,6.00),v60,z5,tPen\WObj:=wPaper;
    MoveL Offs(pOrigin,252.76,29.04,6.00),vTravel,z5,tPen\WObj:=wPaper;
    MoveL Offs(pOrigin,252.76,29.04,0.00),v60,z0,tPen\WObj:=wPaper;
    MoveL Offs(pOrigin,262.23,38.51,0.00),v40,z0,tPen\WObj:=wPaper;
    MoveL Offs(pOrigin,261.87,38.56,0.00),v40,z0,tPen\WObj:=wPaper;
    MoveL Offs(pOrigin,263.97,36.46,0.00),v40,z0,tPen\WObj:=wPaper;
    MoveL Offs(pOrigin,265.02,36.90,0.00),v40,z0,tPen\WObj:=wPaper;
    MoveL Offs(pOrigin,262.76,39.16,0.00),v40,z0,tPen\WObj:=wPaper;
    MoveL Offs(pOrigin,263.39,38.23,0.00),v40,z0,tPen\WObj:=wPaper;
    MoveL Offs(pOrigin,265.73,38.23,0.00),v40,z0,tPen\WObj:=wPaper;
    MoveL Offs(pOrigin,265.91,37.50,0.00),v40,z0,tPen\WObj:=wPaper;
    MoveL Offs(pOrigin,263.81,39.60,0.00),v40,z0,tPen\WObj:=wPaper;
    MoveL Offs(pOrigin,264.93,39.71,0.00),v40,z0,tPen\WObj:=wPaper;
    MoveL Offs(pOrigin,260.87,35.66,0.00),v40,z0,tPen\WObj:=wPaper;
    MoveL Offs(pOrigin,260.98,34.97,0.00),v40,z0,tPen\WObj:=wPaper;
    MoveL Offs(pOrigin,259.02,36.92,0.00),v40,z0,tPen\WObj:=wPaper;
    MoveL Offs(pOrigin,259.77,37.67,0.00),v40,z0,tPen\WObj:=wPaper;
    MoveL Offs(pOrigin,262.03,35.41,0.00),v40,z0,tPen\WObj:=wPaper;
    MoveL Offs(pOrigin,262.92,36.01,0.00),v40,z0,tPen\WObj:=wPaper;
    MoveL Offs(pOrigin,260.82,38.11,0.00),v40,fine,tPen\WObj:=wPaper;
    MoveL Offs(pOrigin,260.82,38.11,6.00),v60,z5,tPen\WObj:=wPaper;
    MoveL Offs(pOrigin,257.98,36.47,6.00),vTravel,z5,tPen\WObj:=wPaper;
    MoveL Offs(pOrigin,257.98,36.47,0.00),v60,z0,tPen\WObj:=wPaper;
    MoveL Offs(pOrigin,260.08,34.37,0.00),v40,z0,tPen\WObj:=wPaper;
    MoveL Offs(pOrigin,259.48,33.47,0.00),v40,z0,tPen\WObj:=wPaper;
    MoveL Offs(pOrigin,257.08,35.88,0.00),v40,z0,tPen\WObj:=wPaper;
    MoveL Offs(pOrigin,257.65,35.06,0.00),v40,z0,tPen\WObj:=wPaper;
    MoveL Offs(pOrigin,259.14,35.06,0.00),v40,fine,tPen\WObj:=wPaper;
    MoveL Offs(pOrigin,259.14,35.06,6.00),v60,z5,tPen\WObj:=wPaper;
    MoveL Offs(pOrigin,256.18,35.28,6.00),vTravel,z5,tPen\WObj:=wPaper;
    MoveL Offs(pOrigin,256.18,35.28,0.00),v60,z0,tPen\WObj:=wPaper;
    MoveL Offs(pOrigin,259.94,31.52,0.00),v40,z0,tPen\WObj:=wPaper;
    MoveL Offs(pOrigin,259.19,30.78,0.00),v40,z0,tPen\WObj:=wPaper;
  ENDPROC

  PROC DrawPart17()
    MoveL Offs(pOrigin,270.01,19.96,0.00),v40,z0,tPen\WObj:=wPaper;
    MoveL Offs(pOrigin,269.36,20.25,0.00),v40,z0,tPen\WObj:=wPaper;
    MoveL Offs(pOrigin,272.37,23.26,0.00),v40,fine,tPen\WObj:=wPaper;
    MoveL Offs(pOrigin,272.37,23.26,6.00),v60,z5,tPen\WObj:=wPaper;
    MoveL Offs(pOrigin,273.71,21.62,6.00),vTravel,z5,tPen\WObj:=wPaper;
    MoveL Offs(pOrigin,273.71,21.62,0.00),v60,z0,tPen\WObj:=wPaper;
    MoveL Offs(pOrigin,277.32,25.22,0.00),v40,z0,tPen\WObj:=wPaper;
    MoveL Offs(pOrigin,277.78,25.63,0.00),v40,z0,tPen\WObj:=wPaper;
    MoveL Offs(pOrigin,281.39,22.02,0.00),v40,z0,tPen\WObj:=wPaper;
    MoveL Offs(pOrigin,280.45,22.39,0.00),v40,z0,tPen\WObj:=wPaper;
    MoveL Offs(pOrigin,282.56,24.49,0.00),v40,z0,tPen\WObj:=wPaper;
    MoveL Offs(pOrigin,282.88,25.01,0.00),v40,z0,tPen\WObj:=wPaper;
    MoveL Offs(pOrigin,285.58,22.31,0.00),v40,z0,tPen\WObj:=wPaper;
    MoveL Offs(pOrigin,285.40,22.85,0.00),v40,z0,tPen\WObj:=wPaper;
    MoveL Offs(pOrigin,288.10,25.56,0.00),v40,z0,tPen\WObj:=wPaper;
    MoveL Offs(pOrigin,288.12,25.75,0.00),v40,z0,tPen\WObj:=wPaper;
    MoveL Offs(pOrigin,290.52,23.34,0.00),v40,z0,tPen\WObj:=wPaper;
    MoveL Offs(pOrigin,291.57,23.79,0.00),v40,z0,tPen\WObj:=wPaper;
    MoveL Offs(pOrigin,289.17,26.19,0.00),v40,fine,tPen\WObj:=wPaper;
    MoveL Offs(pOrigin,289.17,26.19,6.00),v60,z5,tPen\WObj:=wPaper;
    MoveL Offs(pOrigin,290.59,25.56,6.00),vTravel,z5,tPen\WObj:=wPaper;
    MoveL Offs(pOrigin,290.59,25.56,0.00),v60,z0,tPen\WObj:=wPaper;
    MoveL Offs(pOrigin,298.24,25.56,0.00),v40,z0,tPen\WObj:=wPaper;
    MoveL Offs(pOrigin,297.69,26.18,0.00),v40,z0,tPen\WObj:=wPaper;
    MoveL Offs(pOrigin,296.04,24.53,0.00),v40,z0,tPen\WObj:=wPaper;
    MoveL Offs(pOrigin,296.07,23.77,0.00),v40,z0,tPen\WObj:=wPaper;
    MoveL Offs(pOrigin,292.61,27.23,0.00),v40,z0,tPen\WObj:=wPaper;
    MoveL Offs(pOrigin,292.30,26.77,0.00),v40,z0,tPen\WObj:=wPaper;
    MoveL Offs(pOrigin,289.29,23.76,0.00),v40,z0,tPen\WObj:=wPaper;
    MoveL Offs(pOrigin,289.33,23.05,0.00),v40,z0,tPen\WObj:=wPaper;
    MoveL Offs(pOrigin,286.77,25.60,0.00),v40,z0,tPen\WObj:=wPaper;
    MoveL Offs(pOrigin,286.55,24.50,0.00),v40,z0,tPen\WObj:=wPaper;
    MoveL Offs(pOrigin,290.80,24.50,0.00),v40,z0,tPen\WObj:=wPaper;
    MoveL Offs(pOrigin,291.39,24.37,0.00),v40,z0,tPen\WObj:=wPaper;
    MoveL Offs(pOrigin,294.70,27.67,0.00),v40,z0,tPen\WObj:=wPaper;
    MoveL Offs(pOrigin,294.70,28.12,0.00),v40,z0,tPen\WObj:=wPaper;
    MoveL Offs(pOrigin,299.21,23.61,0.00),v40,z0,tPen\WObj:=wPaper;
    MoveL Offs(pOrigin,298.88,24.39,0.00),v40,z0,tPen\WObj:=wPaper;
    MoveL Offs(pOrigin,300.69,26.19,0.00),v40,z0,tPen\WObj:=wPaper;
    MoveL Offs(pOrigin,300.70,26.61,0.00),v40,z0,tPen\WObj:=wPaper;
    MoveL Offs(pOrigin,303.56,23.75,0.00),v40,z0,tPen\WObj:=wPaper;
    MoveL Offs(pOrigin,303.38,24.40,0.00),v40,z0,tPen\WObj:=wPaper;
    MoveL Offs(pOrigin,305.63,26.66,0.00),v40,z0,tPen\WObj:=wPaper;
    MoveL Offs(pOrigin,306.09,27.19,0.00),v40,z0,tPen\WObj:=wPaper;
    MoveL Offs(pOrigin,308.65,24.63,0.00),v40,z0,tPen\WObj:=wPaper;
    MoveL Offs(pOrigin,309.69,25.08,0.00),v40,z0,tPen\WObj:=wPaper;
    MoveL Offs(pOrigin,307.14,27.63,0.00),v40,fine,tPen\WObj:=wPaper;
    MoveL Offs(pOrigin,307.14,27.63,6.00),v60,z5,tPen\WObj:=wPaper;
    MoveL Offs(pOrigin,308.34,27.93,6.00),vTravel,z5,tPen\WObj:=wPaper;
    MoveL Offs(pOrigin,308.34,27.93,0.00),v60,z0,tPen\WObj:=wPaper;
    MoveL Offs(pOrigin,310.74,25.53,0.00),v40,fine,tPen\WObj:=wPaper;
    MoveL Offs(pOrigin,310.74,25.53,6.00),v60,z5,tPen\WObj:=wPaper;
    MoveL Offs(pOrigin,312.09,25.67,6.00),vTravel,z5,tPen\WObj:=wPaper;
    MoveL Offs(pOrigin,312.09,25.67,0.00),v60,z0,tPen\WObj:=wPaper;
    MoveL Offs(pOrigin,309.53,28.23,0.00),v40,z0,tPen\WObj:=wPaper;
    MoveL Offs(pOrigin,310.13,28.17,0.00),v40,z0,tPen\WObj:=wPaper;
    MoveL Offs(pOrigin,306.98,25.01,0.00),v40,z0,tPen\WObj:=wPaper;
    MoveL Offs(pOrigin,307.30,24.49,0.00),v40,z0,tPen\WObj:=wPaper;
    MoveL Offs(pOrigin,304.89,26.89,0.00),v40,z0,tPen\WObj:=wPaper;
    MoveL Offs(pOrigin,303.83,26.35,0.00),v40,z0,tPen\WObj:=wPaper;
    MoveL Offs(pOrigin,301.88,24.40,0.00),v40,z0,tPen\WObj:=wPaper;
    MoveL Offs(pOrigin,302.21,23.60,0.00),v40,z0,tPen\WObj:=wPaper;
    MoveL Offs(pOrigin,299.20,26.61,0.00),v40,z0,tPen\WObj:=wPaper;
    MoveL Offs(pOrigin,299.19,26.19,0.00),v40,z0,tPen\WObj:=wPaper;
    MoveL Offs(pOrigin,297.39,24.39,0.00),v40,z0,tPen\WObj:=wPaper;
    MoveL Offs(pOrigin,297.71,23.62,0.00),v40,z0,tPen\WObj:=wPaper;
    MoveL Offs(pOrigin,293.66,27.68,0.00),v40,z0,tPen\WObj:=wPaper;
    MoveL Offs(pOrigin,293.56,26.62,0.00),v40,z0,tPen\WObj:=wPaper;
    MoveL Offs(pOrigin,295.69,26.62,0.00),v40,z0,tPen\WObj:=wPaper;
    MoveL Offs(pOrigin,295.48,26.67,0.00),v40,z0,tPen\WObj:=wPaper;
    MoveL Offs(pOrigin,295.69,27.10,0.00),v40,z0,tPen\WObj:=wPaper;
    MoveL Offs(pOrigin,295.48,26.67,0.00),v40,z0,tPen\WObj:=wPaper;
    MoveL Offs(pOrigin,295.90,27.52,0.00),v40,z0,tPen\WObj:=wPaper;
    MoveL Offs(pOrigin,286.98,24.76,0.00),v40,z0,tPen\WObj:=wPaper;
    MoveL Offs(pOrigin,283.58,24.12,0.00),v40,z0,tPen\WObj:=wPaper;
    MoveL Offs(pOrigin,279.33,24.12,0.00),v40,z0,tPen\WObj:=wPaper;
    MoveL Offs(pOrigin,276.77,25.19,0.00),v40,z0,tPen\WObj:=wPaper;
    MoveL Offs(pOrigin,274.93,27.74,0.00),v40,z0,tPen\WObj:=wPaper;
    MoveL Offs(pOrigin,274.44,29.44,0.00),v40,z0,tPen\WObj:=wPaper;
    MoveL Offs(pOrigin,275.08,30.15,0.00),v40,z0,tPen\WObj:=wPaper;
    MoveL Offs(pOrigin,280.60,31.92,0.00),v40,z0,tPen\WObj:=wPaper;
    MoveL Offs(pOrigin,289.74,35.95,0.00),v40,z0,tPen\WObj:=wPaper;
    MoveL Offs(pOrigin,293.92,37.37,0.00),v40,z0,tPen\WObj:=wPaper;
    MoveL Offs(pOrigin,294.34,37.94,0.00),v40,z0,tPen\WObj:=wPaper;
    MoveL Offs(pOrigin,294.20,38.29,0.00),v40,z0,tPen\WObj:=wPaper;
    MoveL Offs(pOrigin,292.08,38.01,0.00),v40,z0,tPen\WObj:=wPaper;
    MoveL Offs(pOrigin,291.86,39.64,0.00),v40,z0,tPen\WObj:=wPaper;
    MoveL Offs(pOrigin,292.04,39.95,0.00),v40,z0,tPen\WObj:=wPaper;
    MoveL Offs(pOrigin,286.18,34.09,0.00),v40,z0,tPen\WObj:=wPaper;
    MoveL Offs(pOrigin,286.30,33.54,0.00),v40,z0,tPen\WObj:=wPaper;
    MoveL Offs(pOrigin,284.04,35.79,0.00),v40,z0,tPen\WObj:=wPaper;
    MoveL Offs(pOrigin,284.85,35.06,0.00),v40,z0,tPen\WObj:=wPaper;
    MoveL Offs(pOrigin,287.61,35.06,0.00),v40,z0,tPen\WObj:=wPaper;
    MoveL Offs(pOrigin,287.35,33.99,0.00),v40,z0,tPen\WObj:=wPaper;
    MoveL Offs(pOrigin,284.49,36.84,0.00),v40,fine,tPen\WObj:=wPaper;
    MoveL Offs(pOrigin,284.49,36.84,6.00),v60,z5,tPen\WObj:=wPaper;
    MoveL Offs(pOrigin,285.70,36.24,6.00),vTravel,z5,tPen\WObj:=wPaper;
    MoveL Offs(pOrigin,285.70,36.24,0.00),v60,z0,tPen\WObj:=wPaper;
    MoveL Offs(pOrigin,286.76,36.24,0.00),v40,z0,tPen\WObj:=wPaper;
    MoveL Offs(pOrigin,287.40,36.66,0.00),v40,z0,tPen\WObj:=wPaper;
    MoveL Offs(pOrigin,287.40,36.66,0.00),v40,z0,tPen\WObj:=wPaper;
    MoveL Offs(pOrigin,288.67,36.59,0.00),v40,z0,tPen\WObj:=wPaper;
    MoveL Offs(pOrigin,289.52,37.09,0.00),v40,z0,tPen\WObj:=wPaper;
    MoveL Offs(pOrigin,289.74,37.72,0.00),v40,z0,tPen\WObj:=wPaper;
    MoveL Offs(pOrigin,289.74,37.72,0.00),v40,z0,tPen\WObj:=wPaper;
    MoveL Offs(pOrigin,289.10,37.94,0.00),v40,z0,tPen\WObj:=wPaper;
    MoveL Offs(pOrigin,287.40,36.66,0.00),v40,z0,tPen\WObj:=wPaper;
    MoveL Offs(pOrigin,286.98,36.66,0.00),v40,z0,tPen\WObj:=wPaper;
    MoveL Offs(pOrigin,286.48,37.30,0.00),v40,z0,tPen\WObj:=wPaper;
    MoveL Offs(pOrigin,286.34,38.36,0.00),v40,z0,tPen\WObj:=wPaper;
    MoveL Offs(pOrigin,287.19,39.42,0.00),v40,z0,tPen\WObj:=wPaper;
    MoveL Offs(pOrigin,287.19,39.42,0.00),v40,z0,tPen\WObj:=wPaper;
    MoveL Offs(pOrigin,286.34,38.79,0.00),v40,fine,tPen\WObj:=wPaper;
    MoveL Offs(pOrigin,286.34,38.79,6.00),v60,z5,tPen\WObj:=wPaper;
    MoveL Offs(pOrigin,285.15,39.03,6.00),vTravel,z5,tPen\WObj:=wPaper;
    MoveL Offs(pOrigin,285.15,39.03,0.00),v60,z0,tPen\WObj:=wPaper;
    MoveL Offs(pOrigin,290.56,44.44,0.00),v40,z0,tPen\WObj:=wPaper;
    MoveL Offs(pOrigin,290.91,45.36,0.00),v40,z0,tPen\WObj:=wPaper;
    MoveL Offs(pOrigin,287.00,49.27,0.00),v40,fine,tPen\WObj:=wPaper;
    MoveL Offs(pOrigin,287.00,49.27,6.00),v60,z5,tPen\WObj:=wPaper;
  ENDPROC

  PROC DrawPart18()
    MoveL Offs(pOrigin,284.75,48.53,6.00),vTravel,z5,tPen\WObj:=wPaper;
    MoveL Offs(pOrigin,284.75,48.53,0.00),v60,z0,tPen\WObj:=wPaper;
    MoveL Offs(pOrigin,292.42,40.86,0.00),v40,z0,tPen\WObj:=wPaper;
    MoveL Offs(pOrigin,291.59,41.00,0.00),v40,z0,tPen\WObj:=wPaper;
    MoveL Offs(pOrigin,283.63,33.03,0.00),v40,z0,tPen\WObj:=wPaper;
    MoveL Offs(pOrigin,284.35,32.50,0.00),v40,z0,tPen\WObj:=wPaper;
    MoveL Offs(pOrigin,281.95,34.90,0.00),v40,z0,tPen\WObj:=wPaper;
    MoveL Offs(pOrigin,281.84,34.22,0.00),v40,z0,tPen\WObj:=wPaper;
    MoveL Offs(pOrigin,278.53,30.92,0.00),v40,z0,tPen\WObj:=wPaper;
    MoveL Offs(pOrigin,278.97,30.42,0.00),v40,z0,tPen\WObj:=wPaper;
    MoveL Offs(pOrigin,276.56,32.82,0.00),v40,z0,tPen\WObj:=wPaper;
    MoveL Offs(pOrigin,277.04,32.41,0.00),v40,z0,tPen\WObj:=wPaper;
    MoveL Offs(pOrigin,267.87,23.25,0.00),v40,z0,tPen\WObj:=wPaper;
    MoveL Offs(pOrigin,268.27,23.70,0.00),v40,z0,tPen\WObj:=wPaper;
    MoveL Offs(pOrigin,265.09,22.85,0.00),v40,z0,tPen\WObj:=wPaper;
    MoveL Offs(pOrigin,265.09,23.49,0.00),v40,z0,tPen\WObj:=wPaper;
    MoveL Offs(pOrigin,268.27,24.34,0.00),v40,fine,tPen\WObj:=wPaper;
    MoveL Offs(pOrigin,268.27,24.34,6.00),v60,z5,tPen\WObj:=wPaper;
    MoveL Offs(pOrigin,268.62,22.50,6.00),vTravel,z5,tPen\WObj:=wPaper;
    MoveL Offs(pOrigin,268.62,22.50,0.00),v60,z0,tPen\WObj:=wPaper;
    MoveL Offs(pOrigin,265.31,19.19,0.00),v40,z0,tPen\WObj:=wPaper;
    MoveL Offs(pOrigin,265.37,18.62,0.00),v40,z0,tPen\WObj:=wPaper;
    MoveL Offs(pOrigin,258.61,25.39,0.00),v40,z0,tPen\WObj:=wPaper;
    MoveL Offs(pOrigin,259.34,25.17,0.00),v40,z0,tPen\WObj:=wPaper;
    MoveL Offs(pOrigin,253.93,19.76,0.00),v40,fine,tPen\WObj:=wPaper;
    MoveL Offs(pOrigin,253.93,19.76,6.00),v60,z5,tPen\WObj:=wPaper;
    MoveL Offs(pOrigin,256.03,20.36,6.00),vTravel,z5,tPen\WObj:=wPaper;
    MoveL Offs(pOrigin,256.03,20.36,0.00),v60,z0,tPen\WObj:=wPaper;
    MoveL Offs(pOrigin,261.29,25.62,0.00),v40,fine,tPen\WObj:=wPaper;
    MoveL Offs(pOrigin,261.29,25.62,6.00),v60,z5,tPen\WObj:=wPaper;
    MoveL Offs(pOrigin,259.81,25.68,6.00),vTravel,z5,tPen\WObj:=wPaper;
    MoveL Offs(pOrigin,259.81,25.68,0.00),v60,z0,tPen\WObj:=wPaper;
    MoveL Offs(pOrigin,266.57,18.92,0.00),v40,fine,tPen\WObj:=wPaper;
    MoveL Offs(pOrigin,266.57,18.92,6.00),v60,z5,tPen\WObj:=wPaper;
    MoveL Offs(pOrigin,267.85,20.28,6.00),vTravel,z5,tPen\WObj:=wPaper;
    MoveL Offs(pOrigin,267.85,20.28,0.00),v60,z0,tPen\WObj:=wPaper;
    MoveL Offs(pOrigin,262.75,20.28,0.00),v40,fine,tPen\WObj:=wPaper;
    MoveL Offs(pOrigin,262.75,20.28,6.00),v60,z5,tPen\WObj:=wPaper;
    MoveL Offs(pOrigin,263.81,19.22,6.00),vTravel,z5,tPen\WObj:=wPaper;
    MoveL Offs(pOrigin,263.81,19.22,0.00),v60,z0,tPen\WObj:=wPaper;
    MoveL Offs(pOrigin,258.71,19.22,0.00),v40,z0,tPen\WObj:=wPaper;
    MoveL Offs(pOrigin,258.42,19.77,0.00),v40,z0,tPen\WObj:=wPaper;
    MoveL Offs(pOrigin,255.42,16.77,0.00),v40,z0,tPen\WObj:=wPaper;
    MoveL Offs(pOrigin,255.74,17.11,0.00),v40,z0,tPen\WObj:=wPaper;
    MoveL Offs(pOrigin,250.42,17.11,0.00),v40,z0,tPen\WObj:=wPaper;
    MoveL Offs(pOrigin,250.63,17.95,0.00),v40,z0,tPen\WObj:=wPaper;
    MoveL Offs(pOrigin,247.32,14.64,0.00),v40,z0,tPen\WObj:=wPaper;
    MoveL Offs(pOrigin,247.56,14.04,0.00),v40,z0,tPen\WObj:=wPaper;
    MoveL Offs(pOrigin,240.80,20.80,0.00),v40,z0,tPen\WObj:=wPaper;
    MoveL Offs(pOrigin,241.35,20.62,0.00),v40,z0,tPen\WObj:=wPaper;
    MoveL Offs(pOrigin,238.49,17.76,0.00),v40,z0,tPen\WObj:=wPaper;
    MoveL Offs(pOrigin,237.74,17.01,0.00),v40,z0,tPen\WObj:=wPaper;
    MoveL Offs(pOrigin,235.34,14.61,0.00),v40,z0,tPen\WObj:=wPaper;
    MoveL Offs(pOrigin,234.59,13.86,0.00),v40,z0,tPen\WObj:=wPaper;
    MoveL Offs(pOrigin,232.18,11.45,0.00),v40,z0,tPen\WObj:=wPaper;
    MoveL Offs(pOrigin,231.54,10.64,0.00),v40,z0,tPen\WObj:=wPaper;
    MoveL Offs(pOrigin,221.93,20.26,0.00),v40,z0,tPen\WObj:=wPaper;
    MoveL Offs(pOrigin,221.27,19.96,0.00),v40,z0,tPen\WObj:=wPaper;
    MoveL Offs(pOrigin,219.77,18.45,0.00),v40,fine,tPen\WObj:=wPaper;
    MoveL Offs(pOrigin,219.77,18.45,6.00),v60,z5,tPen\WObj:=wPaper;
    MoveL Offs(pOrigin,220.97,18.16,6.00),vTravel,z5,tPen\WObj:=wPaper;
    MoveL Offs(pOrigin,220.97,18.16,0.00),v60,z0,tPen\WObj:=wPaper;
    MoveL Offs(pOrigin,222.47,19.66,0.00),v40,fine,tPen\WObj:=wPaper;
    MoveL Offs(pOrigin,222.47,19.66,6.00),v60,z5,tPen\WObj:=wPaper;
    MoveL Offs(pOrigin,223.65,19.22,6.00),vTravel,z5,tPen\WObj:=wPaper;
    MoveL Offs(pOrigin,223.65,19.22,0.00),v60,z0,tPen\WObj:=wPaper;
    MoveL Offs(pOrigin,215.58,19.22,0.00),v40,z0,tPen\WObj:=wPaper;
    MoveL Offs(pOrigin,215.58,18.74,0.00),v40,z0,tPen\WObj:=wPaper;
    MoveL Offs(pOrigin,217.23,20.39,0.00),v40,fine,tPen\WObj:=wPaper;
    MoveL Offs(pOrigin,217.23,20.39,6.00),v60,z5,tPen\WObj:=wPaper;
    MoveL Offs(pOrigin,218.43,20.10,6.00),vTravel,z5,tPen\WObj:=wPaper;
    MoveL Offs(pOrigin,218.43,20.10,0.00),v60,z0,tPen\WObj:=wPaper;
    MoveL Offs(pOrigin,216.93,18.60,0.00),v40,fine,tPen\WObj:=wPaper;
    MoveL Offs(pOrigin,216.93,18.60,6.00),v60,z5,tPen\WObj:=wPaper;
    MoveL Offs(pOrigin,218.27,18.45,6.00),vTravel,z5,tPen\WObj:=wPaper;
    MoveL Offs(pOrigin,218.27,18.45,0.00),v60,z0,tPen\WObj:=wPaper;
    MoveL Offs(pOrigin,219.78,19.95,0.00),v40,z0,tPen\WObj:=wPaper;
    MoveL Offs(pOrigin,220.28,20.41,0.00),v40,z0,tPen\WObj:=wPaper;
    MoveL Offs(pOrigin,229.89,10.79,0.00),v40,z0,tPen\WObj:=wPaper;
    MoveL Offs(pOrigin,229.34,11.59,0.00),v40,z0,tPen\WObj:=wPaper;
    MoveL Offs(pOrigin,233.70,15.95,0.00),v40,fine,tPen\WObj:=wPaper;
    MoveL Offs(pOrigin,233.70,15.95,6.00),v60,z5,tPen\WObj:=wPaper;
    MoveL Offs(pOrigin,233.40,17.15,6.00),vTravel,z5,tPen\WObj:=wPaper;
    MoveL Offs(pOrigin,233.40,17.15,0.00),v60,z0,tPen\WObj:=wPaper;
    MoveL Offs(pOrigin,235.35,19.10,0.00),v40,z0,tPen\WObj:=wPaper;
    MoveL Offs(pOrigin,234.66,19.47,0.00),v40,z0,tPen\WObj:=wPaper;
    MoveL Offs(pOrigin,241.57,12.56,0.00),v40,z0,tPen\WObj:=wPaper;
    MoveL Offs(pOrigin,241.33,13.13,0.00),v40,z0,tPen\WObj:=wPaper;
    MoveL Offs(pOrigin,244.33,16.13,0.00),v40,z0,tPen\WObj:=wPaper;
    MoveL Offs(pOrigin,243.43,16.73,0.00),v40,z0,tPen\WObj:=wPaper;
    MoveL Offs(pOrigin,249.30,22.59,0.00),v40,z0,tPen\WObj:=wPaper;
    MoveL Offs(pOrigin,249.18,22.87,0.00),v40,z0,tPen\WObj:=wPaper;
    MoveL Offs(pOrigin,255.94,16.11,0.00),v40,z0,tPen\WObj:=wPaper;
    MoveL Offs(pOrigin,256.99,16.55,0.00),v40,z0,tPen\WObj:=wPaper;
    MoveL Offs(pOrigin,250.38,23.16,0.00),v40,z0,tPen\WObj:=wPaper;
    MoveL Offs(pOrigin,251.24,23.05,0.00),v40,z0,tPen\WObj:=wPaper;
    MoveL Offs(pOrigin,245.53,17.34,0.00),v40,z0,tPen\WObj:=wPaper;
    MoveL Offs(pOrigin,246.58,16.89,0.00),v40,z0,tPen\WObj:=wPaper;
    MoveL Offs(pOrigin,243.28,13.58,0.00),v40,z0,tPen\WObj:=wPaper;
    MoveL Offs(pOrigin,242.77,12.85,0.00),v40,z0,tPen\WObj:=wPaper;
    MoveL Offs(pOrigin,236.01,19.61,0.00),v40,fine,tPen\WObj:=wPaper;
    MoveL Offs(pOrigin,236.01,19.61,6.00),v60,z5,tPen\WObj:=wPaper;
    MoveL Offs(pOrigin,237.21,19.91,6.00),vTravel,z5,tPen\WObj:=wPaper;
    MoveL Offs(pOrigin,237.21,19.91,0.00),v60,z0,tPen\WObj:=wPaper;
    MoveL Offs(pOrigin,244.12,13.00,0.00),v40,z0,tPen\WObj:=wPaper;
    MoveL Offs(pOrigin,245.17,13.44,0.00),v40,z0,tPen\WObj:=wPaper;
    MoveL Offs(pOrigin,238.25,20.36,0.00),v40,z0,tPen\WObj:=wPaper;
    MoveL Offs(pOrigin,239.25,20.01,0.00),v40,z0,tPen\WObj:=wPaper;
    MoveL Offs(pOrigin,236.55,17.31,0.00),v40,fine,tPen\WObj:=wPaper;
    MoveL Offs(pOrigin,236.55,17.31,6.00),v60,z5,tPen\WObj:=wPaper;
    MoveL Offs(pOrigin,237.46,18.17,6.00),vTravel,z5,tPen\WObj:=wPaper;
    MoveL Offs(pOrigin,237.46,18.17,0.00),v60,z0,tPen\WObj:=wPaper;
    MoveL Offs(pOrigin,225.56,18.17,0.00),v40,fine,tPen\WObj:=wPaper;
    MoveL Offs(pOrigin,225.56,18.17,6.00),v60,z5,tPen\WObj:=wPaper;
    MoveL Offs(pOrigin,225.32,19.52,6.00),vTravel,z5,tPen\WObj:=wPaper;
    MoveL Offs(pOrigin,225.32,19.52,0.00),v60,z0,tPen\WObj:=wPaper;
    MoveL Offs(pOrigin,223.82,18.02,0.00),v40,fine,tPen\WObj:=wPaper;
    MoveL Offs(pOrigin,223.82,18.02,6.00),v60,z5,tPen\WObj:=wPaper;
    MoveL Offs(pOrigin,223.82,19.52,6.00),vTravel,z5,tPen\WObj:=wPaper;
    MoveL Offs(pOrigin,223.82,19.52,0.00),v60,z0,tPen\WObj:=wPaper;
  ENDPROC

  PROC DrawPart19()
    MoveL Offs(pOrigin,222.32,18.01,0.00),v40,fine,tPen\WObj:=wPaper;
    MoveL Offs(pOrigin,222.32,18.01,6.00),v60,z5,tPen\WObj:=wPaper;
    MoveL Offs(pOrigin,222.61,16.82,6.00),vTravel,z5,tPen\WObj:=wPaper;
    MoveL Offs(pOrigin,222.61,16.82,0.00),v60,z0,tPen\WObj:=wPaper;
    MoveL Offs(pOrigin,218.41,12.61,0.00),v40,z0,tPen\WObj:=wPaper;
    MoveL Offs(pOrigin,218.36,11.88,0.00),v40,z0,tPen\WObj:=wPaper;
    MoveL Offs(pOrigin,206.79,23.45,0.00),v40,z0,tPen\WObj:=wPaper;
    MoveL Offs(pOrigin,206.45,23.06,0.00),v40,z0,tPen\WObj:=wPaper;
    MoveL Offs(pOrigin,204.65,21.25,0.00),v40,z0,tPen\WObj:=wPaper;
    MoveL Offs(pOrigin,205.38,21.34,0.00),v40,z0,tPen\WObj:=wPaper;
    MoveL Offs(pOrigin,215.15,21.34,0.00),v40,z0,tPen\WObj:=wPaper;
    MoveL Offs(pOrigin,215.15,20.28,0.00),v40,z0,tPen\WObj:=wPaper;
    MoveL Offs(pOrigin,207.08,20.28,0.00),v40,z0,tPen\WObj:=wPaper;
    MoveL Offs(pOrigin,206.29,19.91,0.00),v40,z0,tPen\WObj:=wPaper;
    MoveL Offs(pOrigin,209.15,22.77,0.00),v40,z0,tPen\WObj:=wPaper;
    MoveL Offs(pOrigin,209.41,22.39,0.00),v40,z0,tPen\WObj:=wPaper;
    MoveL Offs(pOrigin,194.11,22.39,0.00),v40,z0,tPen\WObj:=wPaper;
    MoveL Offs(pOrigin,194.32,22.00,0.00),v40,z0,tPen\WObj:=wPaper;
    MoveL Offs(pOrigin,194.32,15.41,0.00),v40,z0,tPen\WObj:=wPaper;
    MoveL Offs(pOrigin,194.89,14.48,0.00),v40,z0,tPen\WObj:=wPaper;
    MoveL Offs(pOrigin,197.00,16.59,0.00),v40,z0,tPen\WObj:=wPaper;
    MoveL Offs(pOrigin,196.24,16.48,0.00),v40,z0,tPen\WObj:=wPaper;
    MoveL Offs(pOrigin,195.81,18.60,0.00),v40,z0,tPen\WObj:=wPaper;
    MoveL Offs(pOrigin,196.45,21.15,0.00),v40,z0,tPen\WObj:=wPaper;
    MoveL Offs(pOrigin,196.45,21.15,0.00),v40,z0,tPen\WObj:=wPaper;
    MoveL Offs(pOrigin,195.39,20.87,0.00),v40,z0,tPen\WObj:=wPaper;
    MoveL Offs(pOrigin,194.75,19.45,0.00),v40,z0,tPen\WObj:=wPaper;
    MoveL Offs(pOrigin,194.75,17.33,0.00),v40,z0,tPen\WObj:=wPaper;
    MoveL Offs(pOrigin,195.18,16.40,0.00),v40,z0,tPen\WObj:=wPaper;
    MoveL Offs(pOrigin,196.66,16.48,0.00),v40,z0,tPen\WObj:=wPaper;
    MoveL Offs(pOrigin,204.74,15.41,0.00),v40,z0,tPen\WObj:=wPaper;
    MoveL Offs(pOrigin,205.38,14.85,0.00),v40,z0,tPen\WObj:=wPaper;
    MoveL Offs(pOrigin,206.37,14.85,0.00),v40,z0,tPen\WObj:=wPaper;
    MoveL Offs(pOrigin,206.23,17.96,0.00),v40,z0,tPen\WObj:=wPaper;
    MoveL Offs(pOrigin,207.29,21.08,0.00),v40,z0,tPen\WObj:=wPaper;
    MoveL Offs(pOrigin,206.65,21.36,0.00),v40,z0,tPen\WObj:=wPaper;
    MoveL Offs(pOrigin,200.49,21.79,0.00),v40,z0,tPen\WObj:=wPaper;
    MoveL Offs(pOrigin,200.49,21.79,0.00),v40,z0,tPen\WObj:=wPaper;
    MoveL Offs(pOrigin,200.27,21.15,0.00),v40,z0,tPen\WObj:=wPaper;
    MoveL Offs(pOrigin,198.15,21.15,0.00),v40,z0,tPen\WObj:=wPaper;
    MoveL Offs(pOrigin,197.51,21.58,0.00),v40,z0,tPen\WObj:=wPaper;
    MoveL Offs(pOrigin,197.51,21.58,0.00),v40,z0,tPen\WObj:=wPaper;
    MoveL Offs(pOrigin,197.94,22.00,0.00),v40,z0,tPen\WObj:=wPaper;
    MoveL Offs(pOrigin,200.49,21.79,0.00),v40,z0,tPen\WObj:=wPaper;
    MoveL Offs(pOrigin,200.31,21.39,0.00),v40,z0,tPen\WObj:=wPaper;
    MoveL Offs(pOrigin,202.26,23.34,0.00),v40,z0,tPen\WObj:=wPaper;
    MoveL Offs(pOrigin,201.84,23.91,0.00),v40,z0,tPen\WObj:=wPaper;
    MoveL Offs(pOrigin,213.26,12.49,0.00),v40,z0,tPen\WObj:=wPaper;
    MoveL Offs(pOrigin,213.17,13.34,0.00),v40,z0,tPen\WObj:=wPaper;
    MoveL Offs(pOrigin,217.07,17.25,0.00),v40,fine,tPen\WObj:=wPaper;
    MoveL Offs(pOrigin,217.07,17.25,6.00),v60,z5,tPen\WObj:=wPaper;
    MoveL Offs(pOrigin,215.72,17.39,6.00),vTravel,z5,tPen\WObj:=wPaper;
    MoveL Offs(pOrigin,215.72,17.39,0.00),v60,z0,tPen\WObj:=wPaper;
    MoveL Offs(pOrigin,211.67,13.34,0.00),v40,z0,tPen\WObj:=wPaper;
    MoveL Offs(pOrigin,211.46,12.80,0.00),v40,z0,tPen\WObj:=wPaper;
    MoveL Offs(pOrigin,205.45,18.81,0.00),v40,fine,tPen\WObj:=wPaper;
    MoveL Offs(pOrigin,205.45,18.81,6.00),v60,z5,tPen\WObj:=wPaper;
    MoveL Offs(pOrigin,205.31,17.46,6.00),vTravel,z5,tPen\WObj:=wPaper;
    MoveL Offs(pOrigin,205.31,17.46,0.00),v60,z0,tPen\WObj:=wPaper;
    MoveL Offs(pOrigin,210.42,12.35,0.00),v40,z0,tPen\WObj:=wPaper;
    MoveL Offs(pOrigin,209.72,12.88,0.00),v40,z0,tPen\WObj:=wPaper;
    MoveL Offs(pOrigin,214.38,17.54,0.00),v40,fine,tPen\WObj:=wPaper;
    MoveL Offs(pOrigin,214.38,17.54,6.00),v60,z5,tPen\WObj:=wPaper;
    MoveL Offs(pOrigin,214.08,18.74,6.00),vTravel,z5,tPen\WObj:=wPaper;
    MoveL Offs(pOrigin,214.08,18.74,0.00),v60,z0,tPen\WObj:=wPaper;
    MoveL Offs(pOrigin,218.44,23.09,0.00),v40,z0,tPen\WObj:=wPaper;
    MoveL Offs(pOrigin,218.62,23.56,0.00),v40,z0,tPen\WObj:=wPaper;
    MoveL Offs(pOrigin,220.57,21.61,0.00),v40,z0,tPen\WObj:=wPaper;
    MoveL Offs(pOrigin,220.53,22.20,0.00),v40,z0,tPen\WObj:=wPaper;
    MoveL Offs(pOrigin,222.34,24.01,0.00),v40,z0,tPen\WObj:=wPaper;
    MoveL Offs(pOrigin,222.21,24.45,0.00),v40,z0,tPen\WObj:=wPaper;
    MoveL Offs(pOrigin,224.17,22.50,0.00),v40,z0,tPen\WObj:=wPaper;
    MoveL Offs(pOrigin,224.58,23.26,0.00),v40,z0,tPen\WObj:=wPaper;
    MoveL Offs(pOrigin,226.08,24.77,0.00),v40,z0,tPen\WObj:=wPaper;
    MoveL Offs(pOrigin,225.95,25.19,0.00),v40,z0,tPen\WObj:=wPaper;
    MoveL Offs(pOrigin,227.91,23.23,0.00),v40,z0,tPen\WObj:=wPaper;
    MoveL Offs(pOrigin,228.18,23.87,0.00),v40,z0,tPen\WObj:=wPaper;
    MoveL Offs(pOrigin,229.98,25.68,0.00),v40,z0,tPen\WObj:=wPaper;
    MoveL Offs(pOrigin,229.55,26.07,0.00),v40,z0,tPen\WObj:=wPaper;
    MoveL Offs(pOrigin,231.50,24.12,0.00),v40,z0,tPen\WObj:=wPaper;
    MoveL Offs(pOrigin,232.07,24.78,0.00),v40,z0,tPen\WObj:=wPaper;
    MoveL Offs(pOrigin,233.58,26.29,0.00),v40,z0,tPen\WObj:=wPaper;
    MoveL Offs(pOrigin,233.14,26.96,0.00),v40,z0,tPen\WObj:=wPaper;
    MoveL Offs(pOrigin,235.24,24.86,0.00),v40,z0,tPen\WObj:=wPaper;
    MoveL Offs(pOrigin,235.97,25.69,0.00),v40,z0,tPen\WObj:=wPaper;
    MoveL Offs(pOrigin,237.48,27.20,0.00),v40,z0,tPen\WObj:=wPaper;
    MoveL Offs(pOrigin,237.03,27.55,0.00),v40,z0,tPen\WObj:=wPaper;
    MoveL Offs(pOrigin,238.99,25.60,0.00),v40,z0,tPen\WObj:=wPaper;
    MoveL Offs(pOrigin,239.72,26.46,0.00),v40,z0,tPen\WObj:=wPaper;
    MoveL Offs(pOrigin,241.37,28.11,0.00),v40,z0,tPen\WObj:=wPaper;
    MoveL Offs(pOrigin,240.78,28.29,0.00),v40,z0,tPen\WObj:=wPaper;
    MoveL Offs(pOrigin,242.73,26.33,0.00),v40,fine,tPen\WObj:=wPaper;
    MoveL Offs(pOrigin,242.73,26.33,6.00),v60,z5,tPen\WObj:=wPaper;
    MoveL Offs(pOrigin,241.67,26.91,6.00),vTravel,z5,tPen\WObj:=wPaper;
    MoveL Offs(pOrigin,241.67,26.91,0.00),v60,z0,tPen\WObj:=wPaper;
    MoveL Offs(pOrigin,243.02,28.26,0.00),v40,z0,tPen\WObj:=wPaper;
    MoveL Offs(pOrigin,243.17,28.88,0.00),v40,z0,tPen\WObj:=wPaper;
    MoveL Offs(pOrigin,245.12,26.93,0.00),v40,fine,tPen\WObj:=wPaper;
    MoveL Offs(pOrigin,245.12,26.93,6.00),v60,z5,tPen\WObj:=wPaper;
    MoveL Offs(pOrigin,243.93,26.63,6.00),vTravel,z5,tPen\WObj:=wPaper;
    MoveL Offs(pOrigin,243.93,26.63,0.00),v60,z0,tPen\WObj:=wPaper;
    MoveL Offs(pOrigin,241.97,28.58,0.00),v40,fine,tPen\WObj:=wPaper;
    MoveL Offs(pOrigin,241.97,28.58,6.00),v60,z5,tPen\WObj:=wPaper;
    MoveL Offs(pOrigin,243.62,27.37,6.00),vTravel,z5,tPen\WObj:=wPaper;
    MoveL Offs(pOrigin,243.62,27.37,0.00),v60,z0,tPen\WObj:=wPaper;
    MoveL Offs(pOrigin,244.97,28.72,0.00),v40,z0,tPen\WObj:=wPaper;
    MoveL Offs(pOrigin,244.37,29.18,0.00),v40,z0,tPen\WObj:=wPaper;
    MoveL Offs(pOrigin,246.32,27.22,0.00),v40,z0,tPen\WObj:=wPaper;
    MoveL Offs(pOrigin,246.81,28.16,0.00),v40,z0,tPen\WObj:=wPaper;
    MoveL Offs(pOrigin,245.96,27.95,0.00),v40,z0,tPen\WObj:=wPaper;
    MoveL Offs(pOrigin,245.75,28.59,0.00),v40,z0,tPen\WObj:=wPaper;
    MoveL Offs(pOrigin,245.75,28.59,0.00),v40,z0,tPen\WObj:=wPaper;
    MoveL Offs(pOrigin,246.81,28.80,0.00),v40,z0,tPen\WObj:=wPaper;
    MoveL Offs(pOrigin,247.66,28.38,0.00),v40,z0,tPen\WObj:=wPaper;
    MoveL Offs(pOrigin,249.57,28.66,0.00),v40,z0,tPen\WObj:=wPaper;
    MoveL Offs(pOrigin,250.21,29.44,0.00),v40,z0,tPen\WObj:=wPaper;
    MoveL Offs(pOrigin,250.21,29.44,0.00),v40,z0,tPen\WObj:=wPaper;
    MoveL Offs(pOrigin,250.00,29.65,0.00),v40,z0,tPen\WObj:=wPaper;
    MoveL Offs(pOrigin,248.09,29.44,0.00),v40,z0,tPen\WObj:=wPaper;
    MoveL Offs(pOrigin,248.09,29.65,0.00),v40,z0,tPen\WObj:=wPaper;
  ENDPROC

  PROC DrawPart20()
    MoveL Offs(pOrigin,248.09,29.65,0.00),v40,z0,tPen\WObj:=wPaper;
    MoveL Offs(pOrigin,245.75,30.57,0.00),v40,z0,tPen\WObj:=wPaper;
    MoveL Offs(pOrigin,244.55,31.85,0.00),v40,z0,tPen\WObj:=wPaper;
    MoveL Offs(pOrigin,243.98,33.83,0.00),v40,z0,tPen\WObj:=wPaper;
    MoveL Offs(pOrigin,243.20,34.18,0.00),v40,z0,tPen\WObj:=wPaper;
    MoveL Offs(pOrigin,241.78,35.60,0.00),v40,z0,tPen\WObj:=wPaper;
    MoveL Offs(pOrigin,241.29,37.30,0.00),v40,z0,tPen\WObj:=wPaper;
    MoveL Offs(pOrigin,241.50,38.15,0.00),v40,z0,tPen\WObj:=wPaper;
    MoveL Offs(pOrigin,241.29,39.00,0.00),v40,z0,tPen\WObj:=wPaper;
    MoveL Offs(pOrigin,210.48,41.12,0.00),v40,z0,tPen\WObj:=wPaper;
    MoveL Offs(pOrigin,206.65,37.87,0.00),v40,z0,tPen\WObj:=wPaper;
    MoveL Offs(pOrigin,203.04,36.24,0.00),v40,z0,tPen\WObj:=wPaper;
    MoveL Offs(pOrigin,202.61,35.39,0.00),v40,z0,tPen\WObj:=wPaper;
    MoveL Offs(pOrigin,202.61,35.06,0.00),v40,z0,tPen\WObj:=wPaper;
    MoveL Offs(pOrigin,198.58,35.06,0.00),v40,fine,tPen\WObj:=wPaper;
    MoveL Offs(pOrigin,198.58,35.06,6.00),v60,z5,tPen\WObj:=wPaper;
    MoveL Offs(pOrigin,197.94,34.01,6.00),vTravel,z5,tPen\WObj:=wPaper;
    MoveL Offs(pOrigin,197.94,34.01,0.00),v60,z0,tPen\WObj:=wPaper;
    MoveL Offs(pOrigin,201.12,34.01,0.00),v40,z0,tPen\WObj:=wPaper;
    MoveL Offs(pOrigin,200.65,34.33,0.00),v40,z0,tPen\WObj:=wPaper;
    MoveL Offs(pOrigin,200.65,36.66,0.00),v40,z0,tPen\WObj:=wPaper;
    MoveL Offs(pOrigin,201.34,37.18,0.00),v40,z0,tPen\WObj:=wPaper;
    MoveL Offs(pOrigin,205.16,37.18,0.00),v40,z0,tPen\WObj:=wPaper;
    MoveL Offs(pOrigin,205.59,37.51,0.00),v40,z0,tPen\WObj:=wPaper;
    MoveL Offs(pOrigin,206.01,37.72,0.00),v40,z0,tPen\WObj:=wPaper;
    MoveL Offs(pOrigin,205.59,37.51,0.00),v40,z0,tPen\WObj:=wPaper;
    MoveL Offs(pOrigin,206.44,37.94,0.00),v40,z0,tPen\WObj:=wPaper;
    MoveL Offs(pOrigin,207.07,38.36,0.00),v40,z0,tPen\WObj:=wPaper;
    MoveL Offs(pOrigin,206.44,37.94,0.00),v40,z0,tPen\WObj:=wPaper;
    MoveL Offs(pOrigin,207.08,38.23,0.00),v40,z0,tPen\WObj:=wPaper;
    MoveL Offs(pOrigin,204.52,38.23,0.00),v40,z0,tPen\WObj:=wPaper;
    MoveL Offs(pOrigin,204.41,38.93,0.00),v40,z0,tPen\WObj:=wPaper;
    MoveL Offs(pOrigin,197.49,32.02,0.00),v40,z0,tPen\WObj:=wPaper;
    MoveL Offs(pOrigin,197.32,31.42,0.00),v40,z0,tPen\WObj:=wPaper;
    MoveL Offs(pOrigin,194.62,34.12,0.00),v40,z0,tPen\WObj:=wPaper;
    MoveL Offs(pOrigin,194.35,33.36,0.00),v40,z0,tPen\WObj:=wPaper;
    MoveL Offs(pOrigin,192.10,31.10,0.00),v40,z0,tPen\WObj:=wPaper;
    MoveL Offs(pOrigin,192.23,30.53,0.00),v40,z0,tPen\WObj:=wPaper;
    MoveL Offs(pOrigin,189.53,33.24,0.00),v40,z0,tPen\WObj:=wPaper;
    MoveL Offs(pOrigin,189.26,32.74,0.00),v40,z0,tPen\WObj:=wPaper;
    MoveL Offs(pOrigin,187.45,30.94,0.00),v40,z0,tPen\WObj:=wPaper;
    MoveL Offs(pOrigin,188.04,30.25,0.00),v40,z0,tPen\WObj:=wPaper;
    MoveL Offs(pOrigin,185.03,33.25,0.00),v40,z0,tPen\WObj:=wPaper;
    MoveL Offs(pOrigin,184.76,32.73,0.00),v40,z0,tPen\WObj:=wPaper;
    MoveL Offs(pOrigin,183.11,31.08,0.00),v40,z0,tPen\WObj:=wPaper;
    MoveL Offs(pOrigin,183.40,30.41,0.00),v40,z0,tPen\WObj:=wPaper;
    MoveL Offs(pOrigin,180.39,33.42,0.00),v40,z0,tPen\WObj:=wPaper;
    MoveL Offs(pOrigin,180.42,32.86,0.00),v40,z0,tPen\WObj:=wPaper;
    MoveL Offs(pOrigin,178.92,31.36,0.00),v40,z0,tPen\WObj:=wPaper;
    MoveL Offs(pOrigin,178.60,30.73,0.00),v40,z0,tPen\WObj:=wPaper;
    MoveL Offs(pOrigin,175.60,33.73,0.00),v40,z0,tPen\WObj:=wPaper;
    MoveL Offs(pOrigin,175.84,33.05,0.00),v40,z0,tPen\WObj:=wPaper;
    MoveL Offs(pOrigin,175.20,32.62,0.00),v40,z0,tPen\WObj:=wPaper;
    MoveL Offs(pOrigin,170.52,32.62,0.00),v40,z0,tPen\WObj:=wPaper;
    MoveL Offs(pOrigin,164.57,33.69,0.00),v40,z0,tPen\WObj:=wPaper;
    MoveL Offs(pOrigin,160.11,35.74,0.00),v40,z0,tPen\WObj:=wPaper;
    MoveL Offs(pOrigin,157.77,37.30,0.00),v40,z0,tPen\WObj:=wPaper;
    MoveL Offs(pOrigin,157.14,38.36,0.00),v40,z0,tPen\WObj:=wPaper;
    MoveL Offs(pOrigin,157.14,38.36,0.00),v40,z0,tPen\WObj:=wPaper;
    MoveL Offs(pOrigin,156.07,41.55,0.00),v40,fine,tPen\WObj:=wPaper;
    MoveL Offs(pOrigin,156.07,41.55,6.00),v60,z5,tPen\WObj:=wPaper;
    MoveL Offs(pOrigin,154.15,40.24,6.00),vTravel,z5,tPen\WObj:=wPaper;
    MoveL Offs(pOrigin,154.15,40.24,0.00),v60,z0,tPen\WObj:=wPaper;
    MoveL Offs(pOrigin,162.42,31.97,0.00),v40,z0,tPen\WObj:=wPaper;
    MoveL Offs(pOrigin,162.59,32.96,0.00),v40,z0,tPen\WObj:=wPaper;
    MoveL Offs(pOrigin,163.80,34.16,0.00),v40,z0,tPen\WObj:=wPaper;
    MoveL Offs(pOrigin,164.51,34.36,0.00),v40,z0,tPen\WObj:=wPaper;
    MoveL Offs(pOrigin,168.12,30.76,0.00),v40,z0,tPen\WObj:=wPaper;
    MoveL Offs(pOrigin,168.58,31.48,0.00),v40,z0,tPen\WObj:=wPaper;
    MoveL Offs(pOrigin,170.08,32.98,0.00),v40,z0,tPen\WObj:=wPaper;
    MoveL Offs(pOrigin,169.90,33.45,0.00),v40,z0,tPen\WObj:=wPaper;
    MoveL Offs(pOrigin,172.91,30.44,0.00),v40,z0,tPen\WObj:=wPaper;
    MoveL Offs(pOrigin,172.77,31.19,0.00),v40,z0,tPen\WObj:=wPaper;
    MoveL Offs(pOrigin,174.58,33.00,0.00),v40,z0,tPen\WObj:=wPaper;
    MoveL Offs(pOrigin,174.40,33.43,0.00),v40,z0,tPen\WObj:=wPaper;
    MoveL Offs(pOrigin,177.10,30.73,0.00),v40,z0,tPen\WObj:=wPaper;
    MoveL Offs(pOrigin,177.42,31.36,0.00),v40,z0,tPen\WObj:=wPaper;
    MoveL Offs(pOrigin,179.22,33.16,0.00),v40,z0,tPen\WObj:=wPaper;
    MoveL Offs(pOrigin,178.59,33.72,0.00),v40,z0,tPen\WObj:=wPaper;
    MoveL Offs(pOrigin,181.90,30.42,0.00),v40,z0,tPen\WObj:=wPaper;
    MoveL Offs(pOrigin,181.61,31.07,0.00),v40,z0,tPen\WObj:=wPaper;
    MoveL Offs(pOrigin,183.26,32.72,0.00),v40,z0,tPen\WObj:=wPaper;
    MoveL Offs(pOrigin,183.54,33.26,0.00),v40,z0,tPen\WObj:=wPaper;
    MoveL Offs(pOrigin,186.54,30.25,0.00),v40,z0,tPen\WObj:=wPaper;
    MoveL Offs(pOrigin,185.96,30.93,0.00),v40,z0,tPen\WObj:=wPaper;
    MoveL Offs(pOrigin,187.76,32.74,0.00),v40,z0,tPen\WObj:=wPaper;
    MoveL Offs(pOrigin,188.03,33.24,0.00),v40,z0,tPen\WObj:=wPaper;
    MoveL Offs(pOrigin,190.89,30.39,0.00),v40,z0,tPen\WObj:=wPaper;
    MoveL Offs(pOrigin,190.45,30.95,0.00),v40,z0,tPen\WObj:=wPaper;
    MoveL Offs(pOrigin,192.70,33.20,0.00),v40,z0,tPen\WObj:=wPaper;
    MoveL Offs(pOrigin,192.37,33.38,0.00),v40,z0,tPen\WObj:=wPaper;
    MoveL Offs(pOrigin,194.93,30.82,0.00),v40,z0,tPen\WObj:=wPaper;
    MoveL Offs(pOrigin,195.54,31.56,0.00),v40,z0,tPen\WObj:=wPaper;
    MoveL Offs(pOrigin,201.86,37.87,0.00),v40,z0,tPen\WObj:=wPaper;
    MoveL Offs(pOrigin,201.20,38.00,0.00),v40,z0,tPen\WObj:=wPaper;
    MoveL Offs(pOrigin,207.36,31.84,0.00),v40,fine,tPen\WObj:=wPaper;
    MoveL Offs(pOrigin,207.36,31.84,6.00),v60,z5,tPen\WObj:=wPaper;
    MoveL Offs(pOrigin,208.86,31.83,6.00),vTravel,z5,tPen\WObj:=wPaper;
    MoveL Offs(pOrigin,208.86,31.83,0.00),v60,z0,tPen\WObj:=wPaper;
    MoveL Offs(pOrigin,202.40,38.29,0.00),v40,z0,tPen\WObj:=wPaper;
    MoveL Offs(pOrigin,203.44,38.74,0.00),v40,z0,tPen\WObj:=wPaper;
    MoveL Offs(pOrigin,210.36,31.83,0.00),v40,fine,tPen\WObj:=wPaper;
    MoveL Offs(pOrigin,210.36,31.83,6.00),v60,z5,tPen\WObj:=wPaper;
    MoveL Offs(pOrigin,211.85,31.82,6.00),vTravel,z5,tPen\WObj:=wPaper;
    MoveL Offs(pOrigin,211.85,31.82,0.00),v60,z0,tPen\WObj:=wPaper;
    MoveL Offs(pOrigin,207.95,35.73,0.00),v40,fine,tPen\WObj:=wPaper;
    MoveL Offs(pOrigin,207.95,35.73,6.00),v60,z5,tPen\WObj:=wPaper;
    MoveL Offs(pOrigin,209.44,35.72,6.00),vTravel,z5,tPen\WObj:=wPaper;
    MoveL Offs(pOrigin,209.44,35.72,0.00),v60,z0,tPen\WObj:=wPaper;
    MoveL Offs(pOrigin,213.35,31.82,0.00),v40,z0,tPen\WObj:=wPaper;
    MoveL Offs(pOrigin,214.40,32.26,0.00),v40,z0,tPen\WObj:=wPaper;
    MoveL Offs(pOrigin,211.24,35.42,0.00),v40,fine,tPen\WObj:=wPaper;
    MoveL Offs(pOrigin,211.24,35.42,6.00),v60,z5,tPen\WObj:=wPaper;
    MoveL Offs(pOrigin,212.74,35.41,6.00),vTravel,z5,tPen\WObj:=wPaper;
    MoveL Offs(pOrigin,212.74,35.41,0.00),v60,z0,tPen\WObj:=wPaper;
    MoveL Offs(pOrigin,215.45,32.71,0.00),v40,z0,tPen\WObj:=wPaper;
    MoveL Offs(pOrigin,216.49,33.16,0.00),v40,z0,tPen\WObj:=wPaper;
    MoveL Offs(pOrigin,214.24,35.41,0.00),v40,fine,tPen\WObj:=wPaper;
    MoveL Offs(pOrigin,214.24,35.41,6.00),v60,z5,tPen\WObj:=wPaper;
    MoveL Offs(pOrigin,215.74,35.40,6.00),vTravel,z5,tPen\WObj:=wPaper;
  ENDPROC

  PROC DrawPart21()
    MoveL Offs(pOrigin,215.74,35.40,0.00),v60,z0,tPen\WObj:=wPaper;
    MoveL Offs(pOrigin,217.69,33.45,0.00),v40,fine,tPen\WObj:=wPaper;
    MoveL Offs(pOrigin,217.69,33.45,6.00),v60,z5,tPen\WObj:=wPaper;
    MoveL Offs(pOrigin,219.19,33.45,6.00),vTravel,z5,tPen\WObj:=wPaper;
    MoveL Offs(pOrigin,219.19,33.45,0.00),v60,z0,tPen\WObj:=wPaper;
    MoveL Offs(pOrigin,217.24,35.40,0.00),v40,fine,tPen\WObj:=wPaper;
    MoveL Offs(pOrigin,217.24,35.40,6.00),v60,z5,tPen\WObj:=wPaper;
    MoveL Offs(pOrigin,218.88,35.25,6.00),vTravel,z5,tPen\WObj:=wPaper;
    MoveL Offs(pOrigin,218.88,35.25,0.00),v60,z0,tPen\WObj:=wPaper;
    MoveL Offs(pOrigin,220.69,33.44,0.00),v40,fine,tPen\WObj:=wPaper;
    MoveL Offs(pOrigin,220.69,33.44,6.00),v60,z5,tPen\WObj:=wPaper;
    MoveL Offs(pOrigin,222.18,33.44,6.00),vTravel,z5,tPen\WObj:=wPaper;
    MoveL Offs(pOrigin,222.18,33.44,0.00),v60,z0,tPen\WObj:=wPaper;
    MoveL Offs(pOrigin,220.38,35.24,0.00),v40,fine,tPen\WObj:=wPaper;
    MoveL Offs(pOrigin,220.38,35.24,6.00),v60,z5,tPen\WObj:=wPaper;
    MoveL Offs(pOrigin,222.18,34.94,6.00),vTravel,z5,tPen\WObj:=wPaper;
    MoveL Offs(pOrigin,222.18,34.94,0.00),v60,z0,tPen\WObj:=wPaper;
    MoveL Offs(pOrigin,223.68,33.43,0.00),v40,fine,tPen\WObj:=wPaper;
    MoveL Offs(pOrigin,223.68,33.43,6.00),v60,z5,tPen\WObj:=wPaper;
    MoveL Offs(pOrigin,223.68,34.93,6.00),vTravel,z5,tPen\WObj:=wPaper;
    MoveL Offs(pOrigin,223.68,34.93,0.00),v60,z0,tPen\WObj:=wPaper;
    MoveL Offs(pOrigin,225.18,33.43,0.00),v40,fine,tPen\WObj:=wPaper;
    MoveL Offs(pOrigin,225.18,33.43,6.00),v60,z5,tPen\WObj:=wPaper;
    MoveL Offs(pOrigin,225.33,34.78,6.00),vTravel,z5,tPen\WObj:=wPaper;
    MoveL Offs(pOrigin,225.33,34.78,0.00),v60,z0,tPen\WObj:=wPaper;
    MoveL Offs(pOrigin,226.68,33.42,0.00),v40,z0,tPen\WObj:=wPaper;
    MoveL Offs(pOrigin,227.12,34.47,0.00),v40,z0,tPen\WObj:=wPaper;
    MoveL Offs(pOrigin,228.18,33.42,0.00),v40,z0,tPen\WObj:=wPaper;
    MoveL Offs(pOrigin,228.77,34.32,0.00),v40,z0,tPen\WObj:=wPaper;
    MoveL Offs(pOrigin,229.52,33.56,0.00),v40,fine,tPen\WObj:=wPaper;
    MoveL Offs(pOrigin,229.52,33.56,6.00),v60,z5,tPen\WObj:=wPaper;
    MoveL Offs(pOrigin,230.41,38.66,6.00),vTravel,z5,tPen\WObj:=wPaper;
    MoveL Offs(pOrigin,230.41,38.66,0.00),v60,z0,tPen\WObj:=wPaper;
    MoveL Offs(pOrigin,214.63,54.43,0.00),v40,z0,tPen\WObj:=wPaper;
    MoveL Offs(pOrigin,215.53,55.03,0.00),v40,z0,tPen\WObj:=wPaper;
    MoveL Offs(pOrigin,231.91,38.65,0.00),v40,z0,tPen\WObj:=wPaper;
    MoveL Offs(pOrigin,231.67,39.31,0.00),v40,z0,tPen\WObj:=wPaper;
    MoveL Offs(pOrigin,233.62,41.27,0.00),v40,z0,tPen\WObj:=wPaper;
    MoveL Offs(pOrigin,233.39,41.64,0.00),v40,z0,tPen\WObj:=wPaper;
    MoveL Offs(pOrigin,236.85,38.19,0.00),v40,z0,tPen\WObj:=wPaper;
    MoveL Offs(pOrigin,237.36,39.03,0.00),v40,z0,tPen\WObj:=wPaper;
    MoveL Offs(pOrigin,239.47,41.13,0.00),v40,z0,tPen\WObj:=wPaper;
    MoveL Offs(pOrigin,238.74,40.91,0.00),v40,z0,tPen\WObj:=wPaper;
    MoveL Offs(pOrigin,237.68,40.49,0.00),v40,z0,tPen\WObj:=wPaper;
    MoveL Offs(pOrigin,227.69,41.41,0.00),v40,z0,tPen\WObj:=wPaper;
    MoveL Offs(pOrigin,222.45,49.41,0.00),v40,z0,tPen\WObj:=wPaper;
    MoveL Offs(pOrigin,226.84,64.50,0.00),v40,z0,tPen\WObj:=wPaper;
    MoveL Offs(pOrigin,227.26,65.14,0.00),v40,z0,tPen\WObj:=wPaper;
    MoveL Offs(pOrigin,227.26,65.14,0.00),v40,z0,tPen\WObj:=wPaper;
    MoveL Offs(pOrigin,227.83,64.93,0.00),v40,z0,tPen\WObj:=wPaper;
    MoveL Offs(pOrigin,230.45,61.31,0.00),v40,z0,tPen\WObj:=wPaper;
    MoveL Offs(pOrigin,236.61,51.54,0.00),v40,fine,tPen\WObj:=wPaper;
    MoveL Offs(pOrigin,236.61,51.54,6.00),v60,z5,tPen\WObj:=wPaper;
    MoveL Offs(pOrigin,235.61,52.87,6.00),vTravel,z5,tPen\WObj:=wPaper;
    MoveL Offs(pOrigin,235.61,52.87,0.00),v60,z0,tPen\WObj:=wPaper;
    MoveL Offs(pOrigin,233.05,55.42,0.00),v40,fine,tPen\WObj:=wPaper;
    MoveL Offs(pOrigin,233.05,55.42,6.00),v60,z5,tPen\WObj:=wPaper;
    MoveL Offs(pOrigin,233.79,57.67,6.00),vTravel,z5,tPen\WObj:=wPaper;
    MoveL Offs(pOrigin,233.79,57.67,0.00),v60,z0,tPen\WObj:=wPaper;
    MoveL Offs(pOrigin,224.78,66.69,0.00),v40,z0,tPen\WObj:=wPaper;
    MoveL Offs(pOrigin,225.46,67.46,0.00),v40,z0,tPen\WObj:=wPaper;
    MoveL Offs(pOrigin,228.77,70.76,0.00),v40,z0,tPen\WObj:=wPaper;
    MoveL Offs(pOrigin,228.32,70.97,0.00),v40,z0,tPen\WObj:=wPaper;
    MoveL Offs(pOrigin,227.05,70.97,0.00),v40,z0,tPen\WObj:=wPaper;
    MoveL Offs(pOrigin,226.38,71.35,0.00),v40,z0,tPen\WObj:=wPaper;
    MoveL Offs(pOrigin,229.53,74.51,0.00),v40,z0,tPen\WObj:=wPaper;
    MoveL Offs(pOrigin,230.00,74.91,0.00),v40,z0,tPen\WObj:=wPaper;
    MoveL Offs(pOrigin,227.14,77.76,0.00),v40,z0,tPen\WObj:=wPaper;
    MoveL Offs(pOrigin,227.59,77.05,0.00),v40,z0,tPen\WObj:=wPaper;
    MoveL Offs(pOrigin,231.80,81.26,0.00),v40,z0,tPen\WObj:=wPaper;
    MoveL Offs(pOrigin,232.52,81.34,0.00),v40,z0,tPen\WObj:=wPaper;
    MoveL Offs(pOrigin,228.47,85.40,0.00),v40,z0,tPen\WObj:=wPaper;
    MoveL Offs(pOrigin,228.82,85.74,0.00),v40,z0,tPen\WObj:=wPaper;
    MoveL Offs(pOrigin,231.67,88.60,0.00),v40,z0,tPen\WObj:=wPaper;
    MoveL Offs(pOrigin,231.30,88.92,0.00),v40,z0,tPen\WObj:=wPaper;
    MoveL Offs(pOrigin,230.02,88.92,0.00),v40,z0,tPen\WObj:=wPaper;
    MoveL Offs(pOrigin,229.43,89.34,0.00),v40,z0,tPen\WObj:=wPaper;
    MoveL Offs(pOrigin,231.98,91.89,0.00),v40,z0,tPen\WObj:=wPaper;
    MoveL Offs(pOrigin,231.51,92.09,0.00),v40,z0,tPen\WObj:=wPaper;
    MoveL Offs(pOrigin,230.45,92.09,0.00),v40,z0,tPen\WObj:=wPaper;
    MoveL Offs(pOrigin,229.59,92.49,0.00),v40,z0,tPen\WObj:=wPaper;
    MoveL Offs(pOrigin,232.29,95.19,0.00),v40,z0,tPen\WObj:=wPaper;
    MoveL Offs(pOrigin,231.94,95.26,0.00),v40,z0,tPen\WObj:=wPaper;
    MoveL Offs(pOrigin,230.66,95.26,0.00),v40,z0,tPen\WObj:=wPaper;
    MoveL Offs(pOrigin,230.05,95.93,0.00),v40,z0,tPen\WObj:=wPaper;
    MoveL Offs(pOrigin,232.75,98.64,0.00),v40,z0,tPen\WObj:=wPaper;
    MoveL Offs(pOrigin,233.07,98.72,0.00),v40,z0,tPen\WObj:=wPaper;
    MoveL Offs(pOrigin,230.06,101.72,0.00),v40,z0,tPen\WObj:=wPaper;
    MoveL Offs(pOrigin,230.52,102.38,0.00),v40,z0,tPen\WObj:=wPaper;
    MoveL Offs(pOrigin,233.07,104.93,0.00),v40,z0,tPen\WObj:=wPaper;
    MoveL Offs(pOrigin,232.58,104.76,0.00),v40,z0,tPen\WObj:=wPaper;
    MoveL Offs(pOrigin,231.51,104.76,0.00),v40,z0,tPen\WObj:=wPaper;
    MoveL Offs(pOrigin,230.82,104.17,0.00),v40,z0,tPen\WObj:=wPaper;
    MoveL Offs(pOrigin,233.07,106.43,0.00),v40,z0,tPen\WObj:=wPaper;
    MoveL Offs(pOrigin,232.58,106.87,0.00),v40,z0,tPen\WObj:=wPaper;
    MoveL Offs(pOrigin,231.51,106.87,0.00),v40,z0,tPen\WObj:=wPaper;
    MoveL Offs(pOrigin,230.83,107.17,0.00),v40,z0,tPen\WObj:=wPaper;
    MoveL Offs(pOrigin,233.08,109.42,0.00),v40,z0,tPen\WObj:=wPaper;
    MoveL Offs(pOrigin,232.79,110.04,0.00),v40,z0,tPen\WObj:=wPaper;
    MoveL Offs(pOrigin,231.72,110.04,0.00),v40,z0,tPen\WObj:=wPaper;
    MoveL Offs(pOrigin,230.99,110.32,0.00),v40,z0,tPen\WObj:=wPaper;
    MoveL Offs(pOrigin,233.09,112.42,0.00),v40,z0,tPen\WObj:=wPaper;
    MoveL Offs(pOrigin,232.79,112.15,0.00),v40,z0,tPen\WObj:=wPaper;
    MoveL Offs(pOrigin,231.72,112.15,0.00),v40,z0,tPen\WObj:=wPaper;
    MoveL Offs(pOrigin,230.99,111.81,0.00),v40,z0,tPen\WObj:=wPaper;
    MoveL Offs(pOrigin,233.40,114.22,0.00),v40,z0,tPen\WObj:=wPaper;
    MoveL Offs(pOrigin,233.92,114.29,0.00),v40,z0,tPen\WObj:=wPaper;
    MoveL Offs(pOrigin,230.61,117.60,0.00),v40,z0,tPen\WObj:=wPaper;
    MoveL Offs(pOrigin,231.01,117.81,0.00),v40,z0,tPen\WObj:=wPaper;
    MoveL Offs(pOrigin,233.12,119.91,0.00),v40,z0,tPen\WObj:=wPaper;
    MoveL Offs(pOrigin,232.58,119.54,0.00),v40,z0,tPen\WObj:=wPaper;
    MoveL Offs(pOrigin,231.51,119.54,0.00),v40,z0,tPen\WObj:=wPaper;
    MoveL Offs(pOrigin,231.02,119.30,0.00),v40,z0,tPen\WObj:=wPaper;
    MoveL Offs(pOrigin,233.12,121.41,0.00),v40,z0,tPen\WObj:=wPaper;
    MoveL Offs(pOrigin,232.58,121.66,0.00),v40,z0,tPen\WObj:=wPaper;
    MoveL Offs(pOrigin,231.51,121.66,0.00),v40,z0,tPen\WObj:=wPaper;
    MoveL Offs(pOrigin,230.88,122.15,0.00),v40,z0,tPen\WObj:=wPaper;
    MoveL Offs(pOrigin,232.98,124.25,0.00),v40,z0,tPen\WObj:=wPaper;
    MoveL Offs(pOrigin,232.58,123.77,0.00),v40,z0,tPen\WObj:=wPaper;
    MoveL Offs(pOrigin,231.51,123.77,0.00),v40,z0,tPen\WObj:=wPaper;
  ENDPROC

  PROC DrawPart22()
    MoveL Offs(pOrigin,230.88,123.65,0.00),v40,z0,tPen\WObj:=wPaper;
    MoveL Offs(pOrigin,232.98,125.75,0.00),v40,z0,tPen\WObj:=wPaper;
    MoveL Offs(pOrigin,232.36,125.88,0.00),v40,z0,tPen\WObj:=wPaper;
    MoveL Offs(pOrigin,231.30,125.88,0.00),v40,z0,tPen\WObj:=wPaper;
    MoveL Offs(pOrigin,230.88,125.15,0.00),v40,z0,tPen\WObj:=wPaper;
    MoveL Offs(pOrigin,232.99,127.25,0.00),v40,z0,tPen\WObj:=wPaper;
    MoveL Offs(pOrigin,233.43,126.73,0.00),v40,z0,tPen\WObj:=wPaper;
    MoveL Offs(pOrigin,229.98,130.18,0.00),v40,z0,tPen\WObj:=wPaper;
    MoveL Offs(pOrigin,230.45,130.69,0.00),v40,z0,tPen\WObj:=wPaper;
    MoveL Offs(pOrigin,232.56,132.79,0.00),v40,z0,tPen\WObj:=wPaper;
    MoveL Offs(pOrigin,232.96,133.17,0.00),v40,z0,tPen\WObj:=wPaper;
    MoveL Offs(pOrigin,229.51,136.63,0.00),v40,z0,tPen\WObj:=wPaper;
    MoveL Offs(pOrigin,229.87,136.08,0.00),v40,z0,tPen\WObj:=wPaper;
    MoveL Offs(pOrigin,231.97,138.18,0.00),v40,z0,tPen\WObj:=wPaper;
    MoveL Offs(pOrigin,232.50,138.12,0.00),v40,z0,tPen\WObj:=wPaper;
    MoveL Offs(pOrigin,229.04,141.57,0.00),v40,z0,tPen\WObj:=wPaper;
    MoveL Offs(pOrigin,229.44,141.62,0.00),v40,z0,tPen\WObj:=wPaper;
    MoveL Offs(pOrigin,231.54,143.72,0.00),v40,z0,tPen\WObj:=wPaper;
    MoveL Offs(pOrigin,231.09,143.83,0.00),v40,z0,tPen\WObj:=wPaper;
    MoveL Offs(pOrigin,230.02,143.83,0.00),v40,z0,tPen\WObj:=wPaper;
    MoveL Offs(pOrigin,229.30,144.47,0.00),v40,z0,tPen\WObj:=wPaper;
    MoveL Offs(pOrigin,231.25,146.42,0.00),v40,z0,tPen\WObj:=wPaper;
    MoveL Offs(pOrigin,231.72,146.36,0.00),v40,z0,tPen\WObj:=wPaper;
    MoveL Offs(pOrigin,228.27,149.81,0.00),v40,z0,tPen\WObj:=wPaper;
    MoveL Offs(pOrigin,228.56,149.71,0.00),v40,z0,tPen\WObj:=wPaper;
    MoveL Offs(pOrigin,230.67,151.81,0.00),v40,z0,tPen\WObj:=wPaper;
    MoveL Offs(pOrigin,230.24,151.22,0.00),v40,z0,tPen\WObj:=wPaper;
    MoveL Offs(pOrigin,229.18,151.22,0.00),v40,z0,tPen\WObj:=wPaper;
    MoveL Offs(pOrigin,228.42,151.05,0.00),v40,z0,tPen\WObj:=wPaper;
    MoveL Offs(pOrigin,230.67,153.31,0.00),v40,z0,tPen\WObj:=wPaper;
    MoveL Offs(pOrigin,230.96,153.10,0.00),v40,z0,tPen\WObj:=wPaper;
    MoveL Offs(pOrigin,227.35,156.71,0.00),v40,z0,tPen\WObj:=wPaper;
    MoveL Offs(pOrigin,227.99,156.59,0.00),v40,z0,tPen\WObj:=wPaper;
    MoveL Offs(pOrigin,229.94,158.55,0.00),v40,z0,tPen\WObj:=wPaper;
    MoveL Offs(pOrigin,229.39,158.62,0.00),v40,z0,tPen\WObj:=wPaper;
    MoveL Offs(pOrigin,228.32,158.62,0.00),v40,z0,tPen\WObj:=wPaper;
    MoveL Offs(pOrigin,227.84,157.94,0.00),v40,z0,tPen\WObj:=wPaper;
    MoveL Offs(pOrigin,229.79,159.90,0.00),v40,z0,tPen\WObj:=wPaper;
    MoveL Offs(pOrigin,229.39,159.67,0.00),v40,z0,tPen\WObj:=wPaper;
    MoveL Offs(pOrigin,228.11,159.67,0.00),v40,z0,tPen\WObj:=wPaper;
    MoveL Offs(pOrigin,227.54,159.14,0.00),v40,z0,tPen\WObj:=wPaper;
    MoveL Offs(pOrigin,231.45,163.05,0.00),v40,z0,tPen\WObj:=wPaper;
    MoveL Offs(pOrigin,231.09,162.68,0.00),v40,z0,tPen\WObj:=wPaper;
    MoveL Offs(pOrigin,231.09,163.52,0.00),v40,z0,tPen\WObj:=wPaper;
    MoveL Offs(pOrigin,230.66,163.95,0.00),v40,z0,tPen\WObj:=wPaper;
    MoveL Offs(pOrigin,230.66,163.95,0.00),v40,z0,tPen\WObj:=wPaper;
    MoveL Offs(pOrigin,229.88,166.50,0.00),v40,z0,tPen\WObj:=wPaper;
    MoveL Offs(pOrigin,229.39,167.14,0.00),v40,z0,tPen\WObj:=wPaper;
    MoveL Offs(pOrigin,229.39,167.14,0.00),v40,z0,tPen\WObj:=wPaper;
    MoveL Offs(pOrigin,228.54,171.39,0.00),v40,z0,tPen\WObj:=wPaper;
    MoveL Offs(pOrigin,229.39,175.43,0.00),v40,z0,tPen\WObj:=wPaper;
    MoveL Offs(pOrigin,229.60,178.19,0.00),v40,z0,tPen\WObj:=wPaper;
    MoveL Offs(pOrigin,230.24,179.04,0.00),v40,z0,tPen\WObj:=wPaper;
    MoveL Offs(pOrigin,229.81,178.68,0.00),v40,z0,tPen\WObj:=wPaper;
    MoveL Offs(pOrigin,228.54,178.68,0.00),v40,z0,tPen\WObj:=wPaper;
    MoveL Offs(pOrigin,228.75,179.74,0.00),v40,z0,tPen\WObj:=wPaper;
    MoveL Offs(pOrigin,229.81,179.74,0.00),v40,z0,tPen\WObj:=wPaper;
    MoveL Offs(pOrigin,230.45,179.97,0.00),v40,z0,tPen\WObj:=wPaper;
    MoveL Offs(pOrigin,225.65,175.16,0.00),v40,z0,tPen\WObj:=wPaper;
    MoveL Offs(pOrigin,226.20,175.51,0.00),v40,z0,tPen\WObj:=wPaper;
    MoveL Offs(pOrigin,229.18,175.51,0.00),v40,z0,tPen\WObj:=wPaper;
    MoveL Offs(pOrigin,229.54,174.58,0.00),v40,z0,tPen\WObj:=wPaper;
    MoveL Offs(pOrigin,226.08,171.12,0.00),v40,z0,tPen\WObj:=wPaper;
    MoveL Offs(pOrigin,226.62,171.29,0.00),v40,z0,tPen\WObj:=wPaper;
    MoveL Offs(pOrigin,228.54,171.29,0.00),v40,z0,tPen\WObj:=wPaper;
    MoveL Offs(pOrigin,228.93,170.98,0.00),v40,z0,tPen\WObj:=wPaper;
    MoveL Offs(pOrigin,226.52,168.57,0.00),v40,z0,tPen\WObj:=wPaper;
    MoveL Offs(pOrigin,226.84,169.18,0.00),v40,z0,tPen\WObj:=wPaper;
    MoveL Offs(pOrigin,228.75,169.18,0.00),v40,z0,tPen\WObj:=wPaper;
    MoveL Offs(pOrigin,229.22,169.78,0.00),v40,z0,tPen\WObj:=wPaper;
    MoveL Offs(pOrigin,226.52,167.08,0.00),v40,z0,tPen\WObj:=wPaper;
    MoveL Offs(pOrigin,225.97,167.05,0.00),v40,z0,tPen\WObj:=wPaper;
    MoveL Offs(pOrigin,233.33,159.68,0.00),v40,z0,tPen\WObj:=wPaper;
    MoveL Offs(pOrigin,232.64,159.75,0.00),v40,z0,tPen\WObj:=wPaper;
    MoveL Offs(pOrigin,231.89,159.00,0.00),v40,z0,tPen\WObj:=wPaper;
    MoveL Offs(pOrigin,231.44,160.05,0.00),v40,z0,tPen\WObj:=wPaper;
    MoveL Offs(pOrigin,232.34,160.95,0.00),v40,z0,tPen\WObj:=wPaper;
    MoveL Offs(pOrigin,232.08,160.98,0.00),v40,z0,tPen\WObj:=wPaper;
    MoveL Offs(pOrigin,231.51,161.33,0.00),v40,z0,tPen\WObj:=wPaper;
    MoveL Offs(pOrigin,231.37,160.55,0.00),v40,z0,tPen\WObj:=wPaper;
    MoveL Offs(pOrigin,232.08,160.20,0.00),v40,z0,tPen\WObj:=wPaper;
    MoveL Offs(pOrigin,232.08,160.98,0.00),v40,z0,tPen\WObj:=wPaper;
    MoveL Offs(pOrigin,232.15,160.12,0.00),v40,z0,tPen\WObj:=wPaper;
    MoveL Offs(pOrigin,240.65,138.24,0.00),v40,fine,tPen\WObj:=wPaper;
    MoveL Offs(pOrigin,240.65,138.24,6.00),v60,z5,tPen\WObj:=wPaper;
    MoveL Offs(pOrigin,243.44,137.63,6.00),vTravel,z5,tPen\WObj:=wPaper;
    MoveL Offs(pOrigin,243.44,137.63,0.00),v60,z0,tPen\WObj:=wPaper;
    MoveL Offs(pOrigin,245.69,135.38,0.00),v40,fine,tPen\WObj:=wPaper;
    MoveL Offs(pOrigin,245.69,135.38,6.00),v60,z5,tPen\WObj:=wPaper;
    MoveL Offs(pOrigin,245.54,134.03,6.00),vTravel,z5,tPen\WObj:=wPaper;
    MoveL Offs(pOrigin,245.54,134.03,0.00),v60,z0,tPen\WObj:=wPaper;
    MoveL Offs(pOrigin,243.29,136.28,0.00),v40,fine,tPen\WObj:=wPaper;
    MoveL Offs(pOrigin,243.29,136.28,6.00),v60,z5,tPen\WObj:=wPaper;
    MoveL Offs(pOrigin,244.25,137.02,6.00),vTravel,z5,tPen\WObj:=wPaper;
    MoveL Offs(pOrigin,244.25,137.02,0.00),v60,z0,tPen\WObj:=wPaper;
    MoveL Offs(pOrigin,245.15,137.92,0.00),v40,z0,tPen\WObj:=wPaper;
    MoveL Offs(pOrigin,244.69,138.24,0.00),v40,z0,tPen\WObj:=wPaper;
    MoveL Offs(pOrigin,244.26,137.81,0.00),v40,z0,tPen\WObj:=wPaper;
    MoveL Offs(pOrigin,244.48,136.96,0.00),v40,fine,tPen\WObj:=wPaper;
    MoveL Offs(pOrigin,244.48,136.96,6.00),v60,z5,tPen\WObj:=wPaper;
    MoveL Offs(pOrigin,245.83,138.22,6.00),vTravel,z5,tPen\WObj:=wPaper;
    MoveL Offs(pOrigin,245.83,138.22,0.00),v60,z0,tPen\WObj:=wPaper;
    MoveL Offs(pOrigin,243.43,140.63,0.00),v40,z0,tPen\WObj:=wPaper;
    MoveL Offs(pOrigin,244.26,140.02,0.00),v40,z0,tPen\WObj:=wPaper;
    MoveL Offs(pOrigin,245.31,141.07,0.00),v40,z0,tPen\WObj:=wPaper;
    MoveL Offs(pOrigin,245.82,141.22,0.00),v40,z0,tPen\WObj:=wPaper;
    MoveL Offs(pOrigin,243.72,143.32,0.00),v40,z0,tPen\WObj:=wPaper;
    MoveL Offs(pOrigin,244.42,143.16,0.00),v40,z0,tPen\WObj:=wPaper;
    MoveL Offs(pOrigin,245.62,144.37,0.00),v40,z0,tPen\WObj:=wPaper;
    MoveL Offs(pOrigin,246.11,143.92,0.00),v40,z0,tPen\WObj:=wPaper;
    MoveL Offs(pOrigin,244.01,146.02,0.00),v40,z0,tPen\WObj:=wPaper;
    MoveL Offs(pOrigin,244.88,146.61,0.00),v40,z0,tPen\WObj:=wPaper;
    MoveL Offs(pOrigin,246.23,147.96,0.00),v40,z0,tPen\WObj:=wPaper;
    MoveL Offs(pOrigin,245.96,148.23,0.00),v40,z0,tPen\WObj:=wPaper;
    MoveL Offs(pOrigin,245.68,148.93,0.00),v40,z0,tPen\WObj:=wPaper;
    MoveL Offs(pOrigin,245.11,148.23,0.00),v40,z0,tPen\WObj:=wPaper;
    MoveL Offs(pOrigin,245.32,147.73,0.00),v40,z0,tPen\WObj:=wPaper;
    MoveL Offs(pOrigin,245.96,148.23,0.00),v40,z0,tPen\WObj:=wPaper;
    MoveL Offs(pOrigin,246.70,147.81,0.00),v40,z0,tPen\WObj:=wPaper;
    MoveL Offs(pOrigin,244.45,150.06,0.00),v40,z0,tPen\WObj:=wPaper;
  ENDPROC

  PROC DrawPart23()
    MoveL Offs(pOrigin,245.04,149.76,0.00),v40,z0,tPen\WObj:=wPaper;
    MoveL Offs(pOrigin,246.84,151.56,0.00),v40,z0,tPen\WObj:=wPaper;
    MoveL Offs(pOrigin,246.39,151.84,0.00),v40,z0,tPen\WObj:=wPaper;
    MoveL Offs(pOrigin,246.18,150.56,0.00),v40,z0,tPen\WObj:=wPaper;
    MoveL Offs(pOrigin,246.18,150.56,0.00),v40,z0,tPen\WObj:=wPaper;
    MoveL Offs(pOrigin,246.10,149.50,0.00),v40,z0,tPen\WObj:=wPaper;
    MoveL Offs(pOrigin,245.54,149.22,0.00),v40,z0,tPen\WObj:=wPaper;
    MoveL Offs(pOrigin,245.32,149.93,0.00),v40,z0,tPen\WObj:=wPaper;
    MoveL Offs(pOrigin,245.54,150.56,0.00),v40,z0,tPen\WObj:=wPaper;
    MoveL Offs(pOrigin,245.54,150.56,0.00),v40,z0,tPen\WObj:=wPaper;
    MoveL Offs(pOrigin,245.75,151.84,0.00),v40,z0,tPen\WObj:=wPaper;
    MoveL Offs(pOrigin,245.20,151.40,0.00),v40,z0,tPen\WObj:=wPaper;
    MoveL Offs(pOrigin,246.85,153.06,0.00),v40,z0,tPen\WObj:=wPaper;
    MoveL Offs(pOrigin,246.60,152.69,0.00),v40,z0,tPen\WObj:=wPaper;
    MoveL Offs(pOrigin,247.73,156.51,0.00),v40,z0,tPen\WObj:=wPaper;
    MoveL Offs(pOrigin,250.00,159.49,0.00),v40,z0,tPen\WObj:=wPaper;
    MoveL Offs(pOrigin,252.55,162.25,0.00),v40,z0,tPen\WObj:=wPaper;
    MoveL Offs(pOrigin,257.65,166.71,0.00),v40,z0,tPen\WObj:=wPaper;
    MoveL Offs(pOrigin,259.63,169.05,0.00),v40,z0,tPen\WObj:=wPaper;
    MoveL Offs(pOrigin,260.62,171.39,0.00),v40,z0,tPen\WObj:=wPaper;
    MoveL Offs(pOrigin,261.55,175.21,0.00),v40,z0,tPen\WObj:=wPaper;
    MoveL Offs(pOrigin,274.93,195.19,0.00),v40,z0,tPen\WObj:=wPaper;
    MoveL Offs(pOrigin,280.88,205.39,0.00),v40,z0,tPen\WObj:=wPaper;
    MoveL Offs(pOrigin,285.77,215.38,0.00),v40,z0,tPen\WObj:=wPaper;
    MoveL Offs(pOrigin,287.75,220.69,0.00),v40,z0,tPen\WObj:=wPaper;
    MoveL Offs(pOrigin,288.18,221.11,0.00),v40,z0,tPen\WObj:=wPaper;
    MoveL Offs(pOrigin,288.25,222.18,0.00),v40,z0,tPen\WObj:=wPaper;
    MoveL Offs(pOrigin,288.30,221.75,0.00),v40,z0,tPen\WObj:=wPaper;
    MoveL Offs(pOrigin,288.30,226.64,0.00),v40,z0,tPen\WObj:=wPaper;
    MoveL Offs(pOrigin,287.83,226.85,0.00),v40,z0,tPen\WObj:=wPaper;
    MoveL Offs(pOrigin,288.04,227.27,0.00),v40,z0,tPen\WObj:=wPaper;
    MoveL Offs(pOrigin,287.83,226.85,0.00),v40,z0,tPen\WObj:=wPaper;
    MoveL Offs(pOrigin,288.04,227.26,0.00),v40,z0,tPen\WObj:=wPaper;
    MoveL Offs(pOrigin,289.31,227.26,0.00),v40,z0,tPen\WObj:=wPaper;
    MoveL Offs(pOrigin,289.92,227.49,0.00),v40,z0,tPen\WObj:=wPaper;
    MoveL Offs(pOrigin,283.91,221.48,0.00),v40,z0,tPen\WObj:=wPaper;
    MoveL Offs(pOrigin,283.47,221.55,0.00),v40,z0,tPen\WObj:=wPaper;
    MoveL Offs(pOrigin,290.54,214.48,0.00),v40,z0,tPen\WObj:=wPaper;
    MoveL Offs(pOrigin,290.03,214.16,0.00),v40,z0,tPen\WObj:=wPaper;
    MoveL Offs(pOrigin,287.93,212.05,0.00),v40,z0,tPen\WObj:=wPaper;
    MoveL Offs(pOrigin,287.40,211.65,0.00),v40,z0,tPen\WObj:=wPaper;
    MoveL Offs(pOrigin,290.10,208.94,0.00),v40,z0,tPen\WObj:=wPaper;
    MoveL Offs(pOrigin,289.71,209.36,0.00),v40,z0,tPen\WObj:=wPaper;
    MoveL Offs(pOrigin,287.01,206.66,0.00),v40,z0,tPen\WObj:=wPaper;
    MoveL Offs(pOrigin,286.52,206.56,0.00),v40,z0,tPen\WObj:=wPaper;
    MoveL Offs(pOrigin,289.22,203.85,0.00),v40,z0,tPen\WObj:=wPaper;
    MoveL Offs(pOrigin,288.80,203.97,0.00),v40,z0,tPen\WObj:=wPaper;
    MoveL Offs(pOrigin,285.79,200.96,0.00),v40,z0,tPen\WObj:=wPaper;
    MoveL Offs(pOrigin,285.48,201.62,0.00),v40,z0,tPen\WObj:=wPaper;
    MoveL Offs(pOrigin,299.31,187.79,0.00),v40,z0,tPen\WObj:=wPaper;
    MoveL Offs(pOrigin,300.14,188.42,0.00),v40,z0,tPen\WObj:=wPaper;
    MoveL Offs(pOrigin,301.49,189.78,0.00),v40,z0,tPen\WObj:=wPaper;
    MoveL Offs(pOrigin,301.40,190.18,0.00),v40,z0,tPen\WObj:=wPaper;
    MoveL Offs(pOrigin,307.26,184.32,0.00),v40,z0,tPen\WObj:=wPaper;
    MoveL Offs(pOrigin,307.47,185.30,0.00),v40,z0,tPen\WObj:=wPaper;
    MoveL Offs(pOrigin,308.82,186.65,0.00),v40,z0,tPen\WObj:=wPaper;
    MoveL Offs(pOrigin,308.90,187.17,0.00),v40,z0,tPen\WObj:=wPaper;
    MoveL Offs(pOrigin,313.70,182.36,0.00),v40,z0,tPen\WObj:=wPaper;
    MoveL Offs(pOrigin,314.05,182.92,0.00),v40,z0,tPen\WObj:=wPaper;
    MoveL Offs(pOrigin,315.55,184.43,0.00),v40,z0,tPen\WObj:=wPaper;
    MoveL Offs(pOrigin,315.49,185.05,0.00),v40,z0,tPen\WObj:=wPaper;
    MoveL Offs(pOrigin,321.35,179.19,0.00),v40,fine,tPen\WObj:=wPaper;
    MoveL Offs(pOrigin,321.35,179.19,6.00),v60,z5,tPen\WObj:=wPaper;
    MoveL Offs(pOrigin,321.65,180.38,6.00),vTravel,z5,tPen\WObj:=wPaper;
    MoveL Offs(pOrigin,321.65,180.38,0.00),v60,z0,tPen\WObj:=wPaper;
    MoveL Offs(pOrigin,318.04,183.99,0.00),v40,z0,tPen\WObj:=wPaper;
    MoveL Offs(pOrigin,317.80,183.68,0.00),v40,z0,tPen\WObj:=wPaper;
    MoveL Offs(pOrigin,316.15,182.03,0.00),v40,z0,tPen\WObj:=wPaper;
    MoveL Offs(pOrigin,316.94,181.85,0.00),v40,z0,tPen\WObj:=wPaper;
    MoveL Offs(pOrigin,318.42,181.85,0.00),v40,z0,tPen\WObj:=wPaper;
    MoveL Offs(pOrigin,318.99,181.89,0.00),v40,z0,tPen\WObj:=wPaper;
    MoveL Offs(pOrigin,315.54,178.43,0.00),v40,z0,tPen\WObj:=wPaper;
    MoveL Offs(pOrigin,315.07,178.01,0.00),v40,z0,tPen\WObj:=wPaper;
    MoveL Offs(pOrigin,317.47,175.60,0.00),v40,z0,tPen\WObj:=wPaper;
    MoveL Offs(pOrigin,316.57,174.99,0.00),v40,z0,tPen\WObj:=wPaper;
    MoveL Offs(pOrigin,313.42,171.84,0.00),v40,z0,tPen\WObj:=wPaper;
    MoveL Offs(pOrigin,313.14,172.47,0.00),v40,z0,tPen\WObj:=wPaper;
    MoveL Offs(pOrigin,315.54,170.07,0.00),v40,z0,tPen\WObj:=wPaper;
    MoveL Offs(pOrigin,315.21,170.64,0.00),v40,z0,tPen\WObj:=wPaper;
    MoveL Offs(pOrigin,312.21,167.64,0.00),v40,z0,tPen\WObj:=wPaper;
    MoveL Offs(pOrigin,311.65,167.98,0.00),v40,z0,tPen\WObj:=wPaper;
    MoveL Offs(pOrigin,314.06,165.58,0.00),v40,z0,tPen\WObj:=wPaper;
    MoveL Offs(pOrigin,314.00,166.45,0.00),v40,z0,tPen\WObj:=wPaper;
    MoveL Offs(pOrigin,310.54,162.99,0.00),v40,z0,tPen\WObj:=wPaper;
    MoveL Offs(pOrigin,310.17,163.49,0.00),v40,z0,tPen\WObj:=wPaper;
    MoveL Offs(pOrigin,312.57,161.09,0.00),v40,z0,tPen\WObj:=wPaper;
    MoveL Offs(pOrigin,312.49,161.95,0.00),v40,z0,tPen\WObj:=wPaper;
    MoveL Offs(pOrigin,309.18,158.64,0.00),v40,z0,tPen\WObj:=wPaper;
    MoveL Offs(pOrigin,308.83,158.85,0.00),v40,z0,tPen\WObj:=wPaper;
    MoveL Offs(pOrigin,311.24,156.45,0.00),v40,z0,tPen\WObj:=wPaper;
    MoveL Offs(pOrigin,310.98,157.45,0.00),v40,z0,tPen\WObj:=wPaper;
    MoveL Offs(pOrigin,307.67,154.14,0.00),v40,z0,tPen\WObj:=wPaper;
    MoveL Offs(pOrigin,307.35,154.36,0.00),v40,z0,tPen\WObj:=wPaper;
    MoveL Offs(pOrigin,309.75,151.96,0.00),v40,z0,tPen\WObj:=wPaper;
    MoveL Offs(pOrigin,308.86,152.28,0.00),v40,z0,tPen\WObj:=wPaper;
    MoveL Offs(pOrigin,307.80,152.28,0.00),v40,z0,tPen\WObj:=wPaper;
    MoveL Offs(pOrigin,307.07,152.04,0.00),v40,z0,tPen\WObj:=wPaper;
    MoveL Offs(pOrigin,310.37,155.35,0.00),v40,z0,tPen\WObj:=wPaper;
    MoveL Offs(pOrigin,310.79,155.40,0.00),v40,z0,tPen\WObj:=wPaper;
    MoveL Offs(pOrigin,308.39,157.81,0.00),v40,z0,tPen\WObj:=wPaper;
    MoveL Offs(pOrigin,307.94,156.76,0.00),v40,z0,tPen\WObj:=wPaper;
    MoveL Offs(pOrigin,310.50,154.20,0.00),v40,z0,tPen\WObj:=wPaper;
    MoveL Offs(pOrigin,310.05,153.16,0.00),v40,z0,tPen\WObj:=wPaper;
    MoveL Offs(pOrigin,307.64,155.56,0.00),v40,z0,tPen\WObj:=wPaper;
    MoveL Offs(pOrigin,308.43,156.39,0.00),v40,z0,tPen\WObj:=wPaper;
    MoveL Offs(pOrigin,311.88,159.85,0.00),v40,z0,tPen\WObj:=wPaper;
    MoveL Offs(pOrigin,312.28,159.89,0.00),v40,z0,tPen\WObj:=wPaper;
    MoveL Offs(pOrigin,309.87,162.30,0.00),v40,z0,tPen\WObj:=wPaper;
    MoveL Offs(pOrigin,310.77,161.78,0.00),v40,z0,tPen\WObj:=wPaper;
    MoveL Offs(pOrigin,311.84,161.78,0.00),v40,fine,tPen\WObj:=wPaper;
    MoveL Offs(pOrigin,311.84,161.78,6.00),v60,z5,tPen\WObj:=wPaper;
    MoveL Offs(pOrigin,313.02,162.14,6.00),vTravel,z5,tPen\WObj:=wPaper;
    MoveL Offs(pOrigin,313.02,162.14,0.00),v60,z0,tPen\WObj:=wPaper;
    MoveL Offs(pOrigin,310.61,164.54,0.00),v40,z0,tPen\WObj:=wPaper;
    MoveL Offs(pOrigin,311.45,165.39,0.00),v40,z0,tPen\WObj:=wPaper;
    MoveL Offs(pOrigin,314.61,168.54,0.00),v40,z0,tPen\WObj:=wPaper;
    MoveL Offs(pOrigin,315.09,169.02,0.00),v40,z0,tPen\WObj:=wPaper;
    MoveL Offs(pOrigin,312.69,171.42,0.00),v40,fine,tPen\WObj:=wPaper;
    MoveL Offs(pOrigin,312.69,171.42,6.00),v60,z5,tPen\WObj:=wPaper;
    MoveL Offs(pOrigin,312.39,170.23,6.00),vTravel,z5,tPen\WObj:=wPaper;
  ENDPROC

